REGION Network 12: Bit startu pompy w trybie awaryjnym na soft-startcie - kasowanie / Bit startu pompyw trybie awaryjnym na soft-startcie
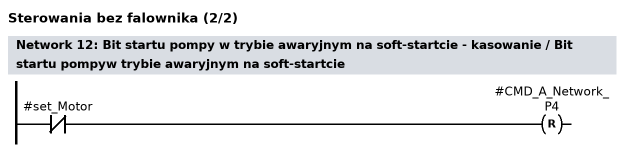
   RUNG wire#powerrail
      I_Contact( #set_Motor )
      R_Coil( #CMD_A_Network_P4 )
   END_RUNG
   // the same network as SCL:
   IF NOT #set_Motor THEN #CMD_A_Network_P4 := FALSE; END_IF;
END_REGION
END_FUNCTION_BLOCK

FUNCTION "Korekta_PV_HWrn_LWrn" : Void
TITLE = Correction
{ S7_Optimized_Access := 'TRUE' }
AUTHOR : rtecmer
VERSION : 0.1
//Funkcja wprowadza korektę ostrzerzeń wysoki i niski poziom wartości procesowej. Wartości te są następnie wykorzystane podczas sterowania pompami dodatkowymi.
   VAR_INPUT 
      PV_HWrn_correction : Real;   // Wspóczninik służący wprowadzeniu korekty ostrzeżenia przekroczenia wartości zadanej bar
      PV_LWrn_correction : Real;   // Wspóczninik służący wprowadzeniu korekty ostrzeżenia zbyt niskia wartości bar w stosunku do zadanej
   END_VAR


BEGIN
	// Funkcja pozwala na wprowadzenie korekty sygnału ostrzeżenia
	// górnrgo i dolnego wartości procesowej
	
	
	
	
	//Przetwornik błąd górny
	"dbdane"."PID_Compact_1_sPid_Cmpt.r_Pv_Hlm" := "dbtags_Sterowanie".SetupControlPompownia.r_Pv_Hlm;
	"PID_Compact_1".sPid_Cmpt.r_Pv_Hlm := "dbdane"."PID_Compact_1_sPid_Cmpt.r_Pv_Hlm";
	
	//Przetwornik błąd dolny
	"dbdane"."PID_Compact_1_sPid_Cmpt.r_Pv_Llm" := "dbtags_Sterowanie".SetupControlPompownia.r_Pv_Llm;
	"PID_Compact_1".sPid_Cmpt.r_Pv_Llm := "dbdane"."PID_Compact_1_sPid_Cmpt.r_Pv_Llm";
	
	//***Wyliczenie ostrzerzeń HWrm i LWrm ***//
	//
	"dbdane"."PID_Compact_1_sPid_Cmpt.r_Pv_HWrn" := ("db10organizacyjna".setpoint_SV_bar + #PV_HWrn_correction);
	"dbdane"."PID_Compact_1_sPid_Cmpt.r_Pv_LWrn" := ("db10organizacyjna".setpoint_SV_bar - #PV_LWrn_correction);
	
	//Ostrzegawczy wysoki
	"PID_Compact_1".sPid_Cmpt.r_Pv_HWrn := "dbdane"."PID_Compact_1_sPid_Cmpt.r_Pv_HWrn";
	"dbtags_Sterowanie".SetupControlPompownia.r_Pv_HWrn := "dbdane"."PID_Compact_1_sPid_Cmpt.r_Pv_HWrn";
	//Ostrzegawczy niski
	"PID_Compact_1".sPid_Cmpt.r_Pv_LWrn := "dbdane"."PID_Compact_1_sPid_Cmpt.r_Pv_LWrn";
	"dbtags_Sterowanie".SetupControlPompownia.r_Pv_LWrn := "dbdane"."PID_Compact_1_sPid_Cmpt.r_Pv_LWrn";
END_FUNCTION

FUNCTION "Synchroniczna_wymiana_danych_PLC1-PLC2" : Void   // FC61, LAD
TITLE = Wymiana danych
{ S7_Optimized_Access := 'TRUE' }
AUTHOR : rtecmer
VERSION : 0.1
// Funkcja grupuje bloki funkcji służąc wymianie danych HMI - PLC1, HMI-PLC2 i SCADA. Wprowadzanie wartości z poziomu HMI Zbiorniki lub HMI Pompownia czy SCADA jest nadpisywane w docelowym sterowniku. Zmian włónych parametrów układu sterowania pompownią, zbiornikami można dokonywać w dowolnego miejsca.
// stored: AutoNumber true, IsIECCheckEnabled false, SetENOAutomatically false, UDAEnableTagReadback false
   VAR_TEMP   // added for the SCL form of the ladder/FBD networks
      _w1 : Bool;
   END_VAR
BEGIN

REGION Network 2: Detekcja zmiany danych - Poziom napełnienia
   // Wymiana danych między PLC 1, PLC 2, SCADA
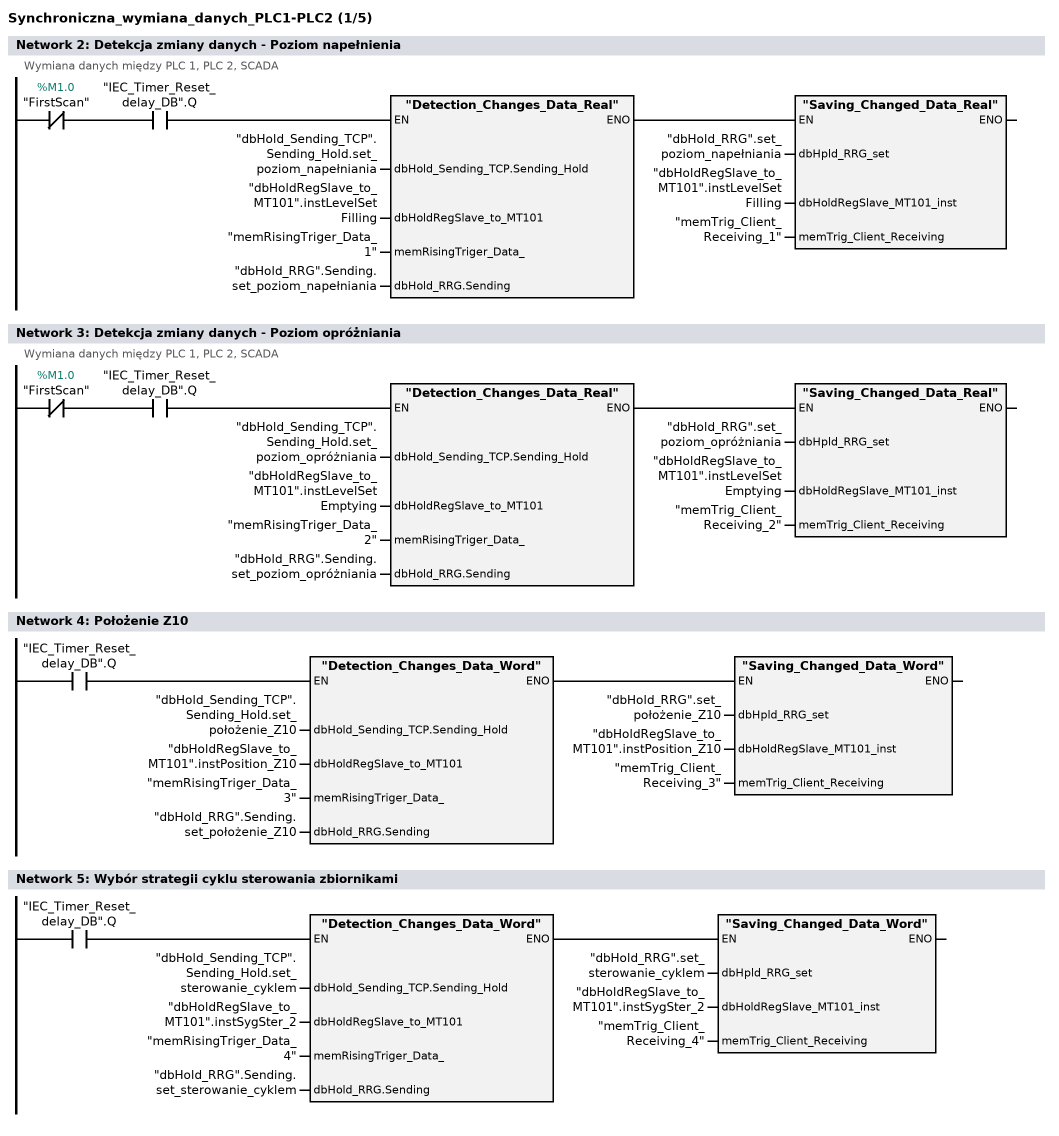
   RUNG wire#powerrail
      I_Contact( "FirstScan" )
      Contact( "IEC_Timer_Reset_delay_DB".Q )
      "Detection_Changes_Data_Real"("dbHold_Sending_TCP.Sending_Hold" := "dbHold_Sending_TCP".Sending_Hold.set_poziom_napełniania, dbHoldRegSlave_to_MT101 := "dbHoldRegSlave_to_MT101".instLevelSetFilling, memRisingTriger_Data_ := "memRisingTriger_Data_1", "dbHold_RRG.Sending" := "dbHold_RRG".Sending.set_poziom_napełniania)
      "Saving_Changed_Data_Real"(dbHpld_RRG_set := "dbHold_RRG".set_poziom_napełniania, dbHoldRegSlave_MT101_inst := "dbHoldRegSlave_to_MT101".instLevelSetFilling, memTrig_Client_Receiving := "memTrig_Client_Receiving_1")
   END_RUNG
   // the same network as SCL:
   "Detection_Changes_Data_Real"(EN := NOT "FirstScan" AND "IEC_Timer_Reset_delay_DB".Q,
                           "dbHold_Sending_TCP.Sending_Hold" := "dbHold_Sending_TCP".Sending_Hold.set_poziom_napełniania,
                           dbHoldRegSlave_to_MT101 := "dbHoldRegSlave_to_MT101".instLevelSetFilling,
                           memRisingTriger_Data_ := "memRisingTriger_Data_1",
                           "dbHold_RRG.Sending" := "dbHold_RRG".Sending.set_poziom_napełniania,
                           ENO => #_w1);
   IF #_w1 THEN
       "Saving_Changed_Data_Real"(dbHpld_RRG_set := "dbHold_RRG".set_poziom_napełniania,
                               dbHoldRegSlave_MT101_inst := "dbHoldRegSlave_to_MT101".instLevelSetFilling,
                               memTrig_Client_Receiving := "memTrig_Client_Receiving_1");
   END_IF;
END_REGION

REGION Network 3: Detekcja zmiany danych - Poziom opróżniania
   // Wymiana danych między PLC 1, PLC 2, SCADA
   RUNG wire#powerrail
      I_Contact( "FirstScan" )
      Contact( "IEC_Timer_Reset_delay_DB".Q )
      "Detection_Changes_Data_Real"("dbHold_Sending_TCP.Sending_Hold" := "dbHold_Sending_TCP".Sending_Hold.set_poziom_opróżniania, dbHoldRegSlave_to_MT101 := "dbHoldRegSlave_to_MT101".instLevelSetEmptying, memRisingTriger_Data_ := "memRisingTriger_Data_2", "dbHold_RRG.Sending" := "dbHold_RRG".Sending.set_poziom_opróżniania)
      "Saving_Changed_Data_Real"(dbHpld_RRG_set := "dbHold_RRG".set_poziom_opróżniania, dbHoldRegSlave_MT101_inst := "dbHoldRegSlave_to_MT101".instLevelSetEmptying, memTrig_Client_Receiving := "memTrig_Client_Receiving_2")
   END_RUNG
   // the same network as SCL:
   "Detection_Changes_Data_Real"(EN := NOT "FirstScan" AND "IEC_Timer_Reset_delay_DB".Q,
                           "dbHold_Sending_TCP.Sending_Hold" := "dbHold_Sending_TCP".Sending_Hold.set_poziom_opróżniania,
                           dbHoldRegSlave_to_MT101 := "dbHoldRegSlave_to_MT101".instLevelSetEmptying,
                           memRisingTriger_Data_ := "memRisingTriger_Data_2",
                           "dbHold_RRG.Sending" := "dbHold_RRG".Sending.set_poziom_opróżniania,
                           ENO => #_w1);
   IF #_w1 THEN
       "Saving_Changed_Data_Real"(dbHpld_RRG_set := "dbHold_RRG".set_poziom_opróżniania,
                               dbHoldRegSlave_MT101_inst := "dbHoldRegSlave_to_MT101".instLevelSetEmptying,
                               memTrig_Client_Receiving := "memTrig_Client_Receiving_2");
   END_IF;
END_REGION

REGION Network 4: Położenie Z10
   RUNG wire#powerrail
      Contact( "IEC_Timer_Reset_delay_DB".Q )
      "Detection_Changes_Data_Word"("dbHold_Sending_TCP.Sending_Hold" := "dbHold_Sending_TCP".Sending_Hold.set_położenie_Z10, dbHoldRegSlave_to_MT101 := "dbHoldRegSlave_to_MT101".instPosition_Z10, memRisingTriger_Data_ := "memRisingTriger_Data_3", "dbHold_RRG.Sending" := "dbHold_RRG".Sending.set_położenie_Z10)
      "Saving_Changed_Data_Word"(dbHpld_RRG_set := "dbHold_RRG".set_położenie_Z10, dbHoldRegSlave_MT101_inst := "dbHoldRegSlave_to_MT101".instPosition_Z10, memTrig_Client_Receiving := "memTrig_Client_Receiving_3")
   END_RUNG
   // the same network as SCL:
   "Detection_Changes_Data_Word"(EN := "IEC_Timer_Reset_delay_DB".Q,
                           "dbHold_Sending_TCP.Sending_Hold" := "dbHold_Sending_TCP".Sending_Hold.set_położenie_Z10,
                           dbHoldRegSlave_to_MT101 := "dbHoldRegSlave_to_MT101".instPosition_Z10,
                           memRisingTriger_Data_ := "memRisingTriger_Data_3",
                           "dbHold_RRG.Sending" := "dbHold_RRG".Sending.set_położenie_Z10,
                           ENO => #_w1);
   IF #_w1 THEN
       "Saving_Changed_Data_Word"(dbHpld_RRG_set := "dbHold_RRG".set_położenie_Z10,
                               dbHoldRegSlave_MT101_inst := "dbHoldRegSlave_to_MT101".instPosition_Z10,
                               memTrig_Client_Receiving := "memTrig_Client_Receiving_3");
   END_IF;
END_REGION

REGION Network 5: Wybór strategii cyklu sterowania zbiornikami
   RUNG wire#powerrail
      Contact( "IEC_Timer_Reset_delay_DB".Q )
      "Detection_Changes_Data_Word"("dbHold_Sending_TCP.Sending_Hold" := "dbHold_Sending_TCP".Sending_Hold.set_sterowanie_cyklem, dbHoldRegSlave_to_MT101 := "dbHoldRegSlave_to_MT101".instSygSter_2, memRisingTriger_Data_ := "memRisingTriger_Data_4", "dbHold_RRG.Sending" := "dbHold_RRG".Sending.set_sterowanie_cyklem)
      "Saving_Changed_Data_Word"(dbHpld_RRG_set := "dbHold_RRG".set_sterowanie_cyklem, dbHoldRegSlave_MT101_inst := "dbHoldRegSlave_to_MT101".instSygSter_2, memTrig_Client_Receiving := "memTrig_Client_Receiving_4")
   END_RUNG
   // the same network as SCL:
   "Detection_Changes_Data_Word"(EN := "IEC_Timer_Reset_delay_DB".Q,
                           "dbHold_Sending_TCP.Sending_Hold" := "dbHold_Sending_TCP".Sending_Hold.set_sterowanie_cyklem,
                           dbHoldRegSlave_to_MT101 := "dbHoldRegSlave_to_MT101".instSygSter_2,
                           memRisingTriger_Data_ := "memRisingTriger_Data_4",
                           "dbHold_RRG.Sending" := "dbHold_RRG".Sending.set_sterowanie_cyklem,
                           ENO => #_w1);
   IF #_w1 THEN
       "Saving_Changed_Data_Word"(dbHpld_RRG_set := "dbHold_RRG".set_sterowanie_cyklem,
                               dbHoldRegSlave_MT101_inst := "dbHoldRegSlave_to_MT101".instSygSter_2,
                               memTrig_Client_Receiving := "memTrig_Client_Receiving_4");
   END_IF;
END_REGION

REGION Network 6: Godzina napełniania start
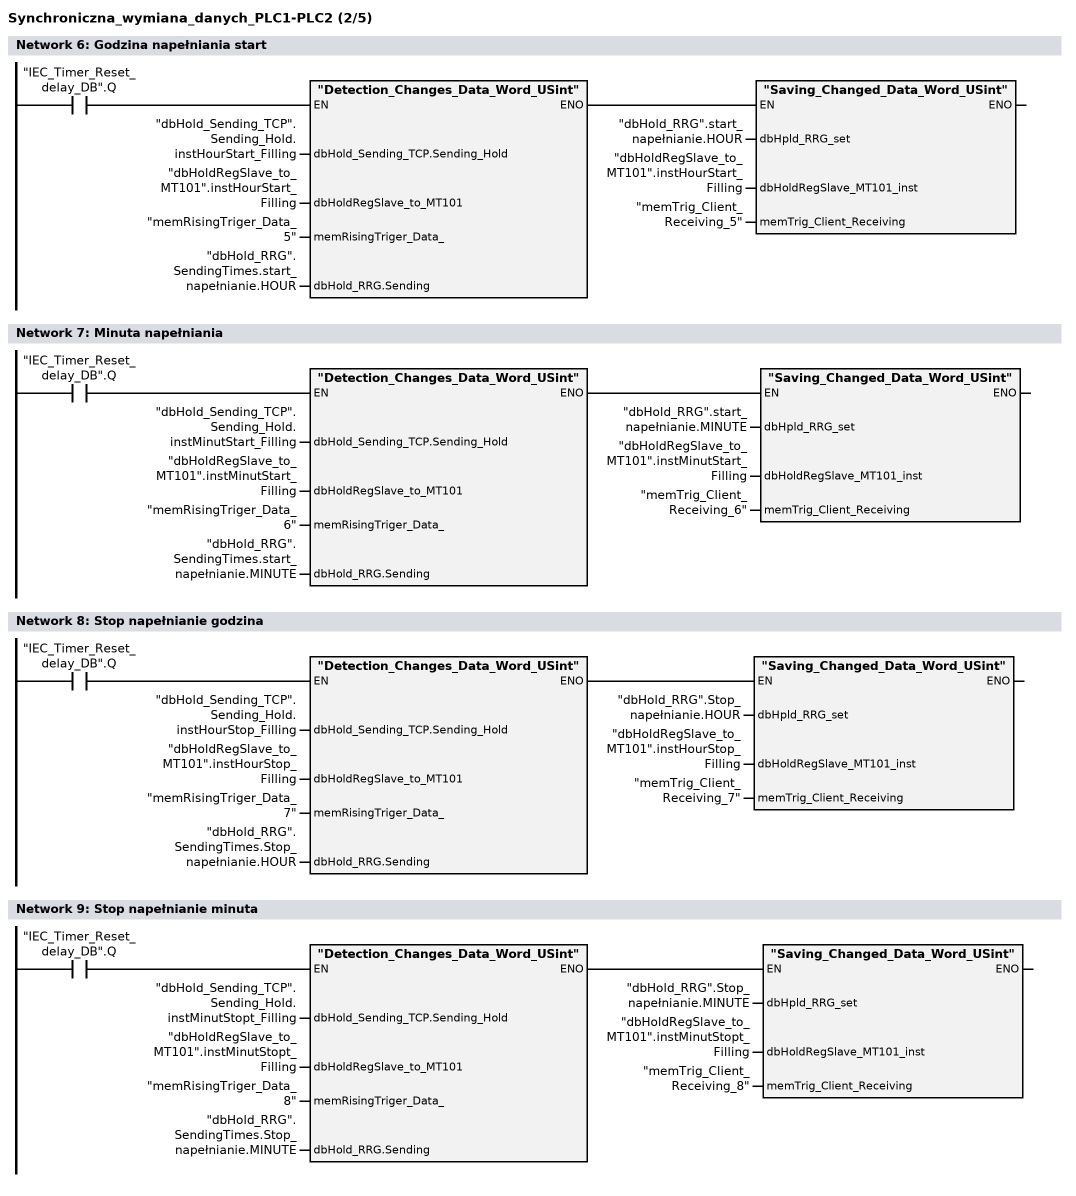
   RUNG wire#powerrail
      Contact( "IEC_Timer_Reset_delay_DB".Q )
      "Detection_Changes_Data_Word_USint"("dbHold_Sending_TCP.Sending_Hold" := "dbHold_Sending_TCP".Sending_Hold.instHourStart_Filling, dbHoldRegSlave_to_MT101 := "dbHoldRegSlave_to_MT101".instHourStart_Filling, memRisingTriger_Data_ := "memRisingTriger_Data_5", "dbHold_RRG.Sending" := "dbHold_RRG".SendingTimes.start_napełnianie.HOUR)
      "Saving_Changed_Data_Word_USint"(dbHpld_RRG_set := "dbHold_RRG".start_napełnianie.HOUR, dbHoldRegSlave_MT101_inst := "dbHoldRegSlave_to_MT101".instHourStart_Filling, memTrig_Client_Receiving := "memTrig_Client_Receiving_5")
   END_RUNG
   // the same network as SCL:
   "Detection_Changes_Data_Word_USint"(EN := "IEC_Timer_Reset_delay_DB".Q,
                           "dbHold_Sending_TCP.Sending_Hold" := "dbHold_Sending_TCP".Sending_Hold.instHourStart_Filling,
                           dbHoldRegSlave_to_MT101 := "dbHoldRegSlave_to_MT101".instHourStart_Filling,
                           memRisingTriger_Data_ := "memRisingTriger_Data_5",
                           "dbHold_RRG.Sending" := "dbHold_RRG".SendingTimes.start_napełnianie.HOUR,
                           ENO => #_w1);
   IF #_w1 THEN
       "Saving_Changed_Data_Word_USint"(dbHpld_RRG_set := "dbHold_RRG".start_napełnianie.HOUR,
                               dbHoldRegSlave_MT101_inst := "dbHoldRegSlave_to_MT101".instHourStart_Filling,
                               memTrig_Client_Receiving := "memTrig_Client_Receiving_5");
   END_IF;
END_REGION

REGION Network 7: Minuta napełniania
   RUNG wire#powerrail
      Contact( "IEC_Timer_Reset_delay_DB".Q )
      "Detection_Changes_Data_Word_USint"("dbHold_Sending_TCP.Sending_Hold" := "dbHold_Sending_TCP".Sending_Hold.instMinutStart_Filling, dbHoldRegSlave_to_MT101 := "dbHoldRegSlave_to_MT101".instMinutStart_Filling, memRisingTriger_Data_ := "memRisingTriger_Data_6", "dbHold_RRG.Sending" := "dbHold_RRG".SendingTimes.start_napełnianie.MINUTE)
      "Saving_Changed_Data_Word_USint"(dbHpld_RRG_set := "dbHold_RRG".start_napełnianie.MINUTE, dbHoldRegSlave_MT101_inst := "dbHoldRegSlave_to_MT101".instMinutStart_Filling, memTrig_Client_Receiving := "memTrig_Client_Receiving_6")
   END_RUNG
   // the same network as SCL:
   "Detection_Changes_Data_Word_USint"(EN := "IEC_Timer_Reset_delay_DB".Q,
                           "dbHold_Sending_TCP.Sending_Hold" := "dbHold_Sending_TCP".Sending_Hold.instMinutStart_Filling,
                           dbHoldRegSlave_to_MT101 := "dbHoldRegSlave_to_MT101".instMinutStart_Filling,
                           memRisingTriger_Data_ := "memRisingTriger_Data_6",
                           "dbHold_RRG.Sending" := "dbHold_RRG".SendingTimes.start_napełnianie.MINUTE,
                           ENO => #_w1);
   IF #_w1 THEN
       "Saving_Changed_Data_Word_USint"(dbHpld_RRG_set := "dbHold_RRG".start_napełnianie.MINUTE,
                               dbHoldRegSlave_MT101_inst := "dbHoldRegSlave_to_MT101".instMinutStart_Filling,
                               memTrig_Client_Receiving := "memTrig_Client_Receiving_6");
   END_IF;
END_REGION

REGION Network 8: Stop napełnianie godzina
   RUNG wire#powerrail
      Contact( "IEC_Timer_Reset_delay_DB".Q )
      "Detection_Changes_Data_Word_USint"("dbHold_Sending_TCP.Sending_Hold" := "dbHold_Sending_TCP".Sending_Hold.instHourStop_Filling, dbHoldRegSlave_to_MT101 := "dbHoldRegSlave_to_MT101".instHourStop_Filling, memRisingTriger_Data_ := "memRisingTriger_Data_7", "dbHold_RRG.Sending" := "dbHold_RRG".SendingTimes.Stop_napełnianie.HOUR)
      "Saving_Changed_Data_Word_USint"(dbHpld_RRG_set := "dbHold_RRG".Stop_napełnianie.HOUR, dbHoldRegSlave_MT101_inst := "dbHoldRegSlave_to_MT101".instHourStop_Filling, memTrig_Client_Receiving := "memTrig_Client_Receiving_7")
   END_RUNG
   // the same network as SCL:
   "Detection_Changes_Data_Word_USint"(EN := "IEC_Timer_Reset_delay_DB".Q,
                           "dbHold_Sending_TCP.Sending_Hold" := "dbHold_Sending_TCP".Sending_Hold.instHourStop_Filling,
                           dbHoldRegSlave_to_MT101 := "dbHoldRegSlave_to_MT101".instHourStop_Filling,
                           memRisingTriger_Data_ := "memRisingTriger_Data_7",
                           "dbHold_RRG.Sending" := "dbHold_RRG".SendingTimes.Stop_napełnianie.HOUR,
                           ENO => #_w1);
   IF #_w1 THEN
       "Saving_Changed_Data_Word_USint"(dbHpld_RRG_set := "dbHold_RRG".Stop_napełnianie.HOUR,
                               dbHoldRegSlave_MT101_inst := "dbHoldRegSlave_to_MT101".instHourStop_Filling,
                               memTrig_Client_Receiving := "memTrig_Client_Receiving_7");
   END_IF;
END_REGION

REGION Network 9: Stop napełnianie minuta
   RUNG wire#powerrail
      Contact( "IEC_Timer_Reset_delay_DB".Q )
      "Detection_Changes_Data_Word_USint"("dbHold_Sending_TCP.Sending_Hold" := "dbHold_Sending_TCP".Sending_Hold.instMinutStopt_Filling, dbHoldRegSlave_to_MT101 := "dbHoldRegSlave_to_MT101".instMinutStopt_Filling, memRisingTriger_Data_ := "memRisingTriger_Data_8", "dbHold_RRG.Sending" := "dbHold_RRG".SendingTimes.Stop_napełnianie.MINUTE)
      "Saving_Changed_Data_Word_USint"(dbHpld_RRG_set := "dbHold_RRG".Stop_napełnianie.MINUTE, dbHoldRegSlave_MT101_inst := "dbHoldRegSlave_to_MT101".instMinutStopt_Filling, memTrig_Client_Receiving := "memTrig_Client_Receiving_8")
   END_RUNG
   // the same network as SCL:
   "Detection_Changes_Data_Word_USint"(EN := "IEC_Timer_Reset_delay_DB".Q,
                           "dbHold_Sending_TCP.Sending_Hold" := "dbHold_Sending_TCP".Sending_Hold.instMinutStopt_Filling,
                           dbHoldRegSlave_to_MT101 := "dbHoldRegSlave_to_MT101".instMinutStopt_Filling,
                           memRisingTriger_Data_ := "memRisingTriger_Data_8",
                           "dbHold_RRG.Sending" := "dbHold_RRG".SendingTimes.Stop_napełnianie.MINUTE,
                           ENO => #_w1);
   IF #_w1 THEN
       "Saving_Changed_Data_Word_USint"(dbHpld_RRG_set := "dbHold_RRG".Stop_napełnianie.MINUTE,
                               dbHoldRegSlave_MT101_inst := "dbHoldRegSlave_to_MT101".instMinutStopt_Filling,
                               memTrig_Client_Receiving := "memTrig_Client_Receiving_8");
   END_IF;
END_REGION

REGION Network 10: Start przetłaczanie (miasto) godzina
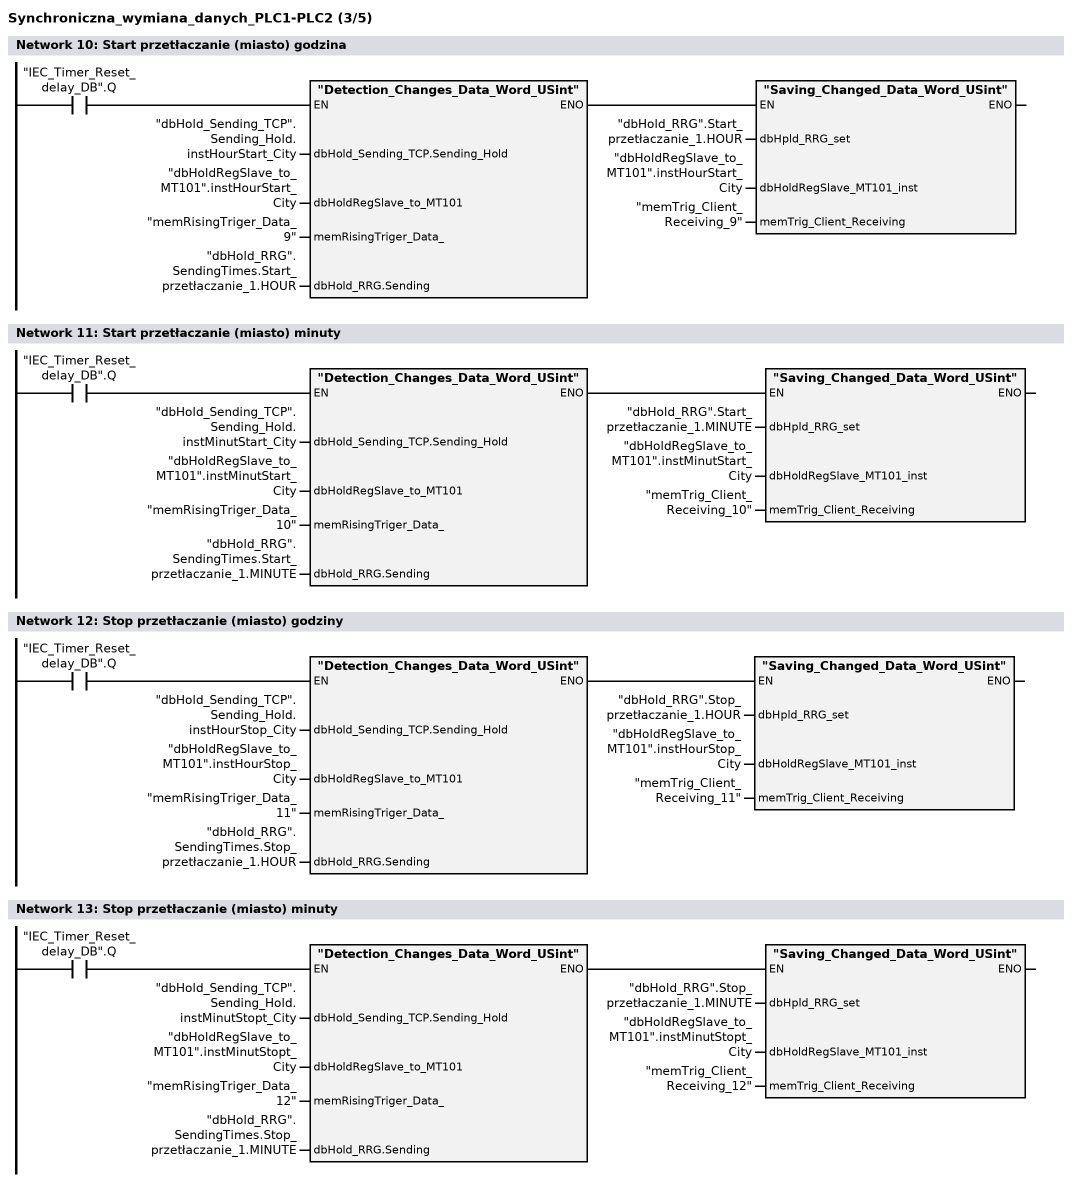
   RUNG wire#powerrail
      Contact( "IEC_Timer_Reset_delay_DB".Q )
      "Detection_Changes_Data_Word_USint"("dbHold_Sending_TCP.Sending_Hold" := "dbHold_Sending_TCP".Sending_Hold.instHourStart_City, dbHoldRegSlave_to_MT101 := "dbHoldRegSlave_to_MT101".instHourStart_City, memRisingTriger_Data_ := "memRisingTriger_Data_9", "dbHold_RRG.Sending" := "dbHold_RRG".SendingTimes.Start_przetłaczanie_1.HOUR)
      "Saving_Changed_Data_Word_USint"(dbHpld_RRG_set := "dbHold_RRG".Start_przetłaczanie_1.HOUR, dbHoldRegSlave_MT101_inst := "dbHoldRegSlave_to_MT101".instHourStart_City, memTrig_Client_Receiving := "memTrig_Client_Receiving_9")
   END_RUNG
   // the same network as SCL:
   "Detection_Changes_Data_Word_USint"(EN := "IEC_Timer_Reset_delay_DB".Q,
                           "dbHold_Sending_TCP.Sending_Hold" := "dbHold_Sending_TCP".Sending_Hold.instHourStart_City,
                           dbHoldRegSlave_to_MT101 := "dbHoldRegSlave_to_MT101".instHourStart_City,
                           memRisingTriger_Data_ := "memRisingTriger_Data_9",
                           "dbHold_RRG.Sending" := "dbHold_RRG".SendingTimes.Start_przetłaczanie_1.HOUR,
                           ENO => #_w1);
   IF #_w1 THEN
       "Saving_Changed_Data_Word_USint"(dbHpld_RRG_set := "dbHold_RRG".Start_przetłaczanie_1.HOUR,
                               dbHoldRegSlave_MT101_inst := "dbHoldRegSlave_to_MT101".instHourStart_City,
                               memTrig_Client_Receiving := "memTrig_Client_Receiving_9");
   END_IF;
END_REGION

REGION Network 11: Start przetłaczanie (miasto) minuty
   RUNG wire#powerrail
      Contact( "IEC_Timer_Reset_delay_DB".Q )
      "Detection_Changes_Data_Word_USint"("dbHold_Sending_TCP.Sending_Hold" := "dbHold_Sending_TCP".Sending_Hold.instMinutStart_City, dbHoldRegSlave_to_MT101 := "dbHoldRegSlave_to_MT101".instMinutStart_City, memRisingTriger_Data_ := "memRisingTriger_Data_10", "dbHold_RRG.Sending" := "dbHold_RRG".SendingTimes.Start_przetłaczanie_1.MINUTE)
      "Saving_Changed_Data_Word_USint"(dbHpld_RRG_set := "dbHold_RRG".Start_przetłaczanie_1.MINUTE, dbHoldRegSlave_MT101_inst := "dbHoldRegSlave_to_MT101".instMinutStart_City, memTrig_Client_Receiving := "memTrig_Client_Receiving_10")
   END_RUNG
   // the same network as SCL:
   "Detection_Changes_Data_Word_USint"(EN := "IEC_Timer_Reset_delay_DB".Q,
                           "dbHold_Sending_TCP.Sending_Hold" := "dbHold_Sending_TCP".Sending_Hold.instMinutStart_City,
                           dbHoldRegSlave_to_MT101 := "dbHoldRegSlave_to_MT101".instMinutStart_City,
                           memRisingTriger_Data_ := "memRisingTriger_Data_10",
                           "dbHold_RRG.Sending" := "dbHold_RRG".SendingTimes.Start_przetłaczanie_1.MINUTE,
                           ENO => #_w1);
   IF #_w1 THEN
       "Saving_Changed_Data_Word_USint"(dbHpld_RRG_set := "dbHold_RRG".Start_przetłaczanie_1.MINUTE,
                               dbHoldRegSlave_MT101_inst := "dbHoldRegSlave_to_MT101".instMinutStart_City,
                               memTrig_Client_Receiving := "memTrig_Client_Receiving_10");
   END_IF;
END_REGION

REGION Network 12: Stop przetłaczanie (miasto) godziny
   RUNG wire#powerrail
      Contact( "IEC_Timer_Reset_delay_DB".Q )
      "Detection_Changes_Data_Word_USint"("dbHold_Sending_TCP.Sending_Hold" := "dbHold_Sending_TCP".Sending_Hold.instHourStop_City, dbHoldRegSlave_to_MT101 := "dbHoldRegSlave_to_MT101".instHourStop_City, memRisingTriger_Data_ := "memRisingTriger_Data_11", "dbHold_RRG.Sending" := "dbHold_RRG".SendingTimes.Stop_przetłaczanie_1.HOUR)
      "Saving_Changed_Data_Word_USint"(dbHpld_RRG_set := "dbHold_RRG".Stop_przetłaczanie_1.HOUR, dbHoldRegSlave_MT101_inst := "dbHoldRegSlave_to_MT101".instHourStop_City, memTrig_Client_Receiving := "memTrig_Client_Receiving_11")
   END_RUNG
   // the same network as SCL:
   "Detection_Changes_Data_Word_USint"(EN := "IEC_Timer_Reset_delay_DB".Q,
                           "dbHold_Sending_TCP.Sending_Hold" := "dbHold_Sending_TCP".Sending_Hold.instHourStop_City,
                           dbHoldRegSlave_to_MT101 := "dbHoldRegSlave_to_MT101".instHourStop_City,
                           memRisingTriger_Data_ := "memRisingTriger_Data_11",
                           "dbHold_RRG.Sending" := "dbHold_RRG".SendingTimes.Stop_przetłaczanie_1.HOUR,
                           ENO => #_w1);
   IF #_w1 THEN
       "Saving_Changed_Data_Word_USint"(dbHpld_RRG_set := "dbHold_RRG".Stop_przetłaczanie_1.HOUR,
                               dbHoldRegSlave_MT101_inst := "dbHoldRegSlave_to_MT101".instHourStop_City,
                               memTrig_Client_Receiving := "memTrig_Client_Receiving_11");
   END_IF;
END_REGION

REGION Network 13: Stop przetłaczanie (miasto) minuty
   RUNG wire#powerrail
      Contact( "IEC_Timer_Reset_delay_DB".Q )
      "Detection_Changes_Data_Word_USint"("dbHold_Sending_TCP.Sending_Hold" := "dbHold_Sending_TCP".Sending_Hold.instMinutStopt_City, dbHoldRegSlave_to_MT101 := "dbHoldRegSlave_to_MT101".instMinutStopt_City, memRisingTriger_Data_ := "memRisingTriger_Data_12", "dbHold_RRG.Sending" := "dbHold_RRG".SendingTimes.Stop_przetłaczanie_1.MINUTE)
      "Saving_Changed_Data_Word_USint"(dbHpld_RRG_set := "dbHold_RRG".Stop_przetłaczanie_1.MINUTE, dbHoldRegSlave_MT101_inst := "dbHoldRegSlave_to_MT101".instMinutStopt_City, memTrig_Client_Receiving := "memTrig_Client_Receiving_12")
   END_RUNG
   // the same network as SCL:
   "Detection_Changes_Data_Word_USint"(EN := "IEC_Timer_Reset_delay_DB".Q,
                           "dbHold_Sending_TCP.Sending_Hold" := "dbHold_Sending_TCP".Sending_Hold.instMinutStopt_City,
                           dbHoldRegSlave_to_MT101 := "dbHoldRegSlave_to_MT101".instMinutStopt_City,
                           memRisingTriger_Data_ := "memRisingTriger_Data_12",
                           "dbHold_RRG.Sending" := "dbHold_RRG".SendingTimes.Stop_przetłaczanie_1.MINUTE,
                           ENO => #_w1);
   IF #_w1 THEN
       "Saving_Changed_Data_Word_USint"(dbHpld_RRG_set := "dbHold_RRG".Stop_przetłaczanie_1.MINUTE,
                               dbHoldRegSlave_MT101_inst := "dbHoldRegSlave_to_MT101".instMinutStopt_City,
                               memTrig_Client_Receiving := "memTrig_Client_Receiving_12");
   END_IF;
END_REGION

REGION Network 14: Start dosilanie godziny
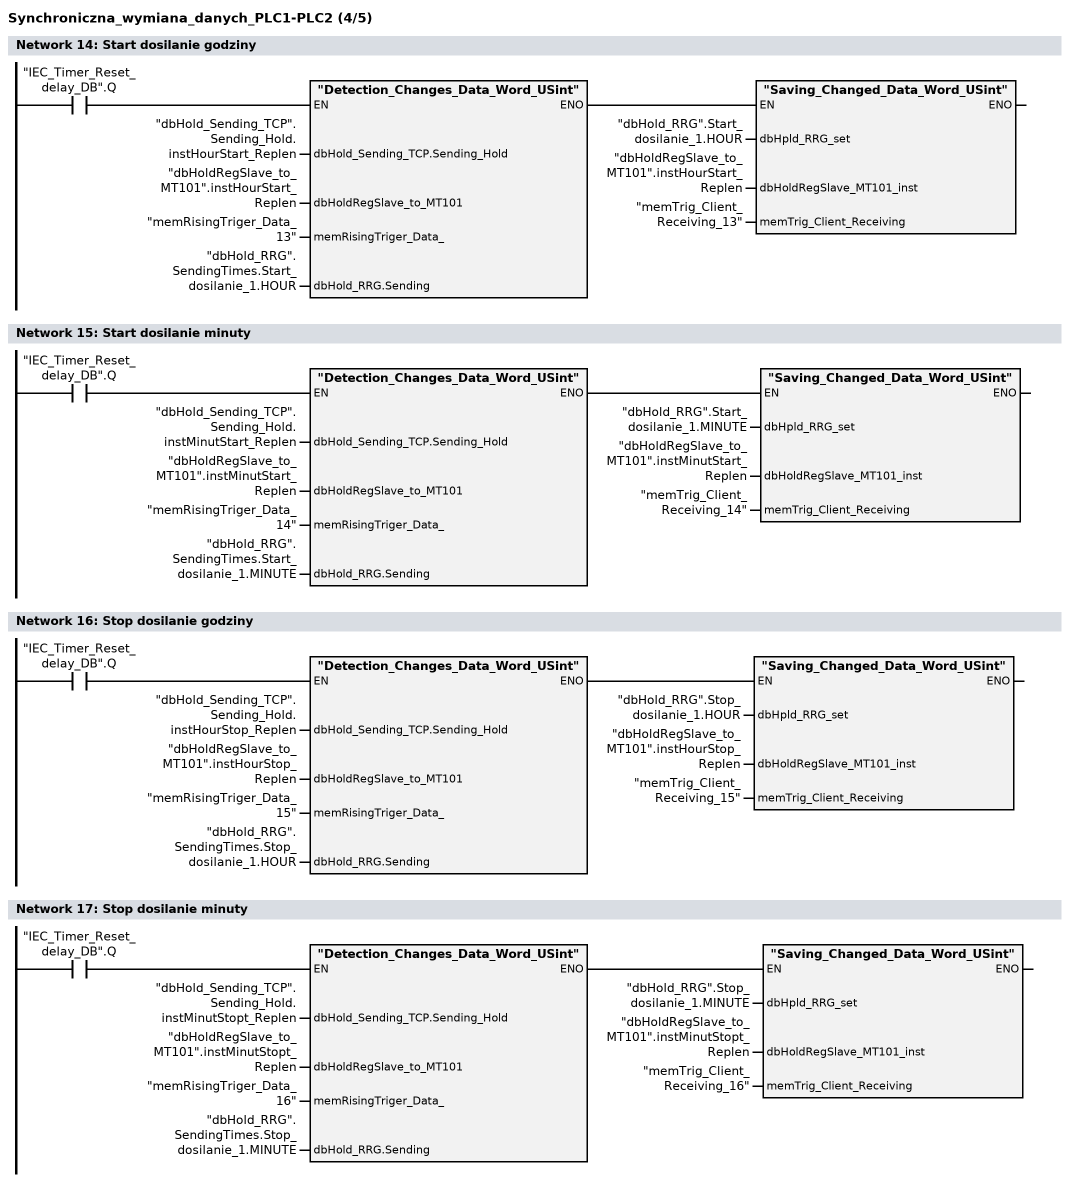
   RUNG wire#powerrail
      Contact( "IEC_Timer_Reset_delay_DB".Q )
      "Detection_Changes_Data_Word_USint"("dbHold_Sending_TCP.Sending_Hold" := "dbHold_Sending_TCP".Sending_Hold.instHourStart_Replen, dbHoldRegSlave_to_MT101 := "dbHoldRegSlave_to_MT101".instHourStart_Replen, memRisingTriger_Data_ := "memRisingTriger_Data_13", "dbHold_RRG.Sending" := "dbHold_RRG".SendingTimes.Start_dosilanie_1.HOUR)
      "Saving_Changed_Data_Word_USint"(dbHpld_RRG_set := "dbHold_RRG".Start_dosilanie_1.HOUR, dbHoldRegSlave_MT101_inst := "dbHoldRegSlave_to_MT101".instHourStart_Replen, memTrig_Client_Receiving := "memTrig_Client_Receiving_13")
   END_RUNG
   // the same network as SCL:
   "Detection_Changes_Data_Word_USint"(EN := "IEC_Timer_Reset_delay_DB".Q,
                           "dbHold_Sending_TCP.Sending_Hold" := "dbHold_Sending_TCP".Sending_Hold.instHourStart_Replen,
                           dbHoldRegSlave_to_MT101 := "dbHoldRegSlave_to_MT101".instHourStart_Replen,
                           memRisingTriger_Data_ := "memRisingTriger_Data_13",
                           "dbHold_RRG.Sending" := "dbHold_RRG".SendingTimes.Start_dosilanie_1.HOUR,
                           ENO => #_w1);
   IF #_w1 THEN
       "Saving_Changed_Data_Word_USint"(dbHpld_RRG_set := "dbHold_RRG".Start_dosilanie_1.HOUR,
                               dbHoldRegSlave_MT101_inst := "dbHoldRegSlave_to_MT101".instHourStart_Replen,
                               memTrig_Client_Receiving := "memTrig_Client_Receiving_13");
   END_IF;
END_REGION

REGION Network 15: Start dosilanie minuty
   RUNG wire#powerrail
      Contact( "IEC_Timer_Reset_delay_DB".Q )
      "Detection_Changes_Data_Word_USint"("dbHold_Sending_TCP.Sending_Hold" := "dbHold_Sending_TCP".Sending_Hold.instMinutStart_Replen, dbHoldRegSlave_to_MT101 := "dbHoldRegSlave_to_MT101".instMinutStart_Replen, memRisingTriger_Data_ := "memRisingTriger_Data_14", "dbHold_RRG.Sending" := "dbHold_RRG".SendingTimes.Start_dosilanie_1.MINUTE)
      "Saving_Changed_Data_Word_USint"(dbHpld_RRG_set := "dbHold_RRG".Start_dosilanie_1.MINUTE, dbHoldRegSlave_MT101_inst := "dbHoldRegSlave_to_MT101".instMinutStart_Replen, memTrig_Client_Receiving := "memTrig_Client_Receiving_14")
   END_RUNG
   // the same network as SCL:
   "Detection_Changes_Data_Word_USint"(EN := "IEC_Timer_Reset_delay_DB".Q,
                           "dbHold_Sending_TCP.Sending_Hold" := "dbHold_Sending_TCP".Sending_Hold.instMinutStart_Replen,
                           dbHoldRegSlave_to_MT101 := "dbHoldRegSlave_to_MT101".instMinutStart_Replen,
                           memRisingTriger_Data_ := "memRisingTriger_Data_14",
                           "dbHold_RRG.Sending" := "dbHold_RRG".SendingTimes.Start_dosilanie_1.MINUTE,
                           ENO => #_w1);
   IF #_w1 THEN
       "Saving_Changed_Data_Word_USint"(dbHpld_RRG_set := "dbHold_RRG".Start_dosilanie_1.MINUTE,
                               dbHoldRegSlave_MT101_inst := "dbHoldRegSlave_to_MT101".instMinutStart_Replen,
                               memTrig_Client_Receiving := "memTrig_Client_Receiving_14");
   END_IF;
END_REGION

REGION Network 16: Stop dosilanie godziny
   RUNG wire#powerrail
      Contact( "IEC_Timer_Reset_delay_DB".Q )
      "Detection_Changes_Data_Word_USint"("dbHold_Sending_TCP.Sending_Hold" := "dbHold_Sending_TCP".Sending_Hold.instHourStop_Replen, dbHoldRegSlave_to_MT101 := "dbHoldRegSlave_to_MT101".instHourStop_Replen, memRisingTriger_Data_ := "memRisingTriger_Data_15", "dbHold_RRG.Sending" := "dbHold_RRG".SendingTimes.Stop_dosilanie_1.HOUR)
      "Saving_Changed_Data_Word_USint"(dbHpld_RRG_set := "dbHold_RRG".Stop_dosilanie_1.HOUR, dbHoldRegSlave_MT101_inst := "dbHoldRegSlave_to_MT101".instHourStop_Replen, memTrig_Client_Receiving := "memTrig_Client_Receiving_15")
   END_RUNG
   // the same network as SCL:
   "Detection_Changes_Data_Word_USint"(EN := "IEC_Timer_Reset_delay_DB".Q,
                           "dbHold_Sending_TCP.Sending_Hold" := "dbHold_Sending_TCP".Sending_Hold.instHourStop_Replen,
                           dbHoldRegSlave_to_MT101 := "dbHoldRegSlave_to_MT101".instHourStop_Replen,
                           memRisingTriger_Data_ := "memRisingTriger_Data_15",
                           "dbHold_RRG.Sending" := "dbHold_RRG".SendingTimes.Stop_dosilanie_1.HOUR,
                           ENO => #_w1);
   IF #_w1 THEN
       "Saving_Changed_Data_Word_USint"(dbHpld_RRG_set := "dbHold_RRG".Stop_dosilanie_1.HOUR,
                               dbHoldRegSlave_MT101_inst := "dbHoldRegSlave_to_MT101".instHourStop_Replen,
                               memTrig_Client_Receiving := "memTrig_Client_Receiving_15");
   END_IF;
END_REGION

REGION Network 17: Stop dosilanie minuty
   RUNG wire#powerrail
      Contact( "IEC_Timer_Reset_delay_DB".Q )
      "Detection_Changes_Data_Word_USint"("dbHold_Sending_TCP.Sending_Hold" := "dbHold_Sending_TCP".Sending_Hold.instMinutStopt_Replen, dbHoldRegSlave_to_MT101 := "dbHoldRegSlave_to_MT101".instMinutStopt_Replen, memRisingTriger_Data_ := "memRisingTriger_Data_16", "dbHold_RRG.Sending" := "dbHold_RRG".SendingTimes.Stop_dosilanie_1.MINUTE)
      "Saving_Changed_Data_Word_USint"(dbHpld_RRG_set := "dbHold_RRG".Stop_dosilanie_1.MINUTE, dbHoldRegSlave_MT101_inst := "dbHoldRegSlave_to_MT101".instMinutStopt_Replen, memTrig_Client_Receiving := "memTrig_Client_Receiving_16")
   END_RUNG
   // the same network as SCL:
   "Detection_Changes_Data_Word_USint"(EN := "IEC_Timer_Reset_delay_DB".Q,
                           "dbHold_Sending_TCP.Sending_Hold" := "dbHold_Sending_TCP".Sending_Hold.instMinutStopt_Replen,
                           dbHoldRegSlave_to_MT101 := "dbHoldRegSlave_to_MT101".instMinutStopt_Replen,
                           memRisingTriger_Data_ := "memRisingTriger_Data_16",
                           "dbHold_RRG.Sending" := "dbHold_RRG".SendingTimes.Stop_dosilanie_1.MINUTE,
                           ENO => #_w1);
   IF #_w1 THEN
       "Saving_Changed_Data_Word_USint"(dbHpld_RRG_set := "dbHold_RRG".Stop_dosilanie_1.MINUTE,
                               dbHoldRegSlave_MT101_inst := "dbHoldRegSlave_to_MT101".instMinutStopt_Replen,
                               memTrig_Client_Receiving := "memTrig_Client_Receiving_16");
   END_IF;
END_REGION

REGION Network 19: Wybór trymu pracy M1,M2,M3,M4, Z1-Z8
   // dbHoldRegSlave_MT101 - tu wartość zadajemy 
   // dbHoldSending_TCP.Sending_Hold - z tą wzmienną porównujemy 
   // dbHold_REG.Sending - tu wysyłamy
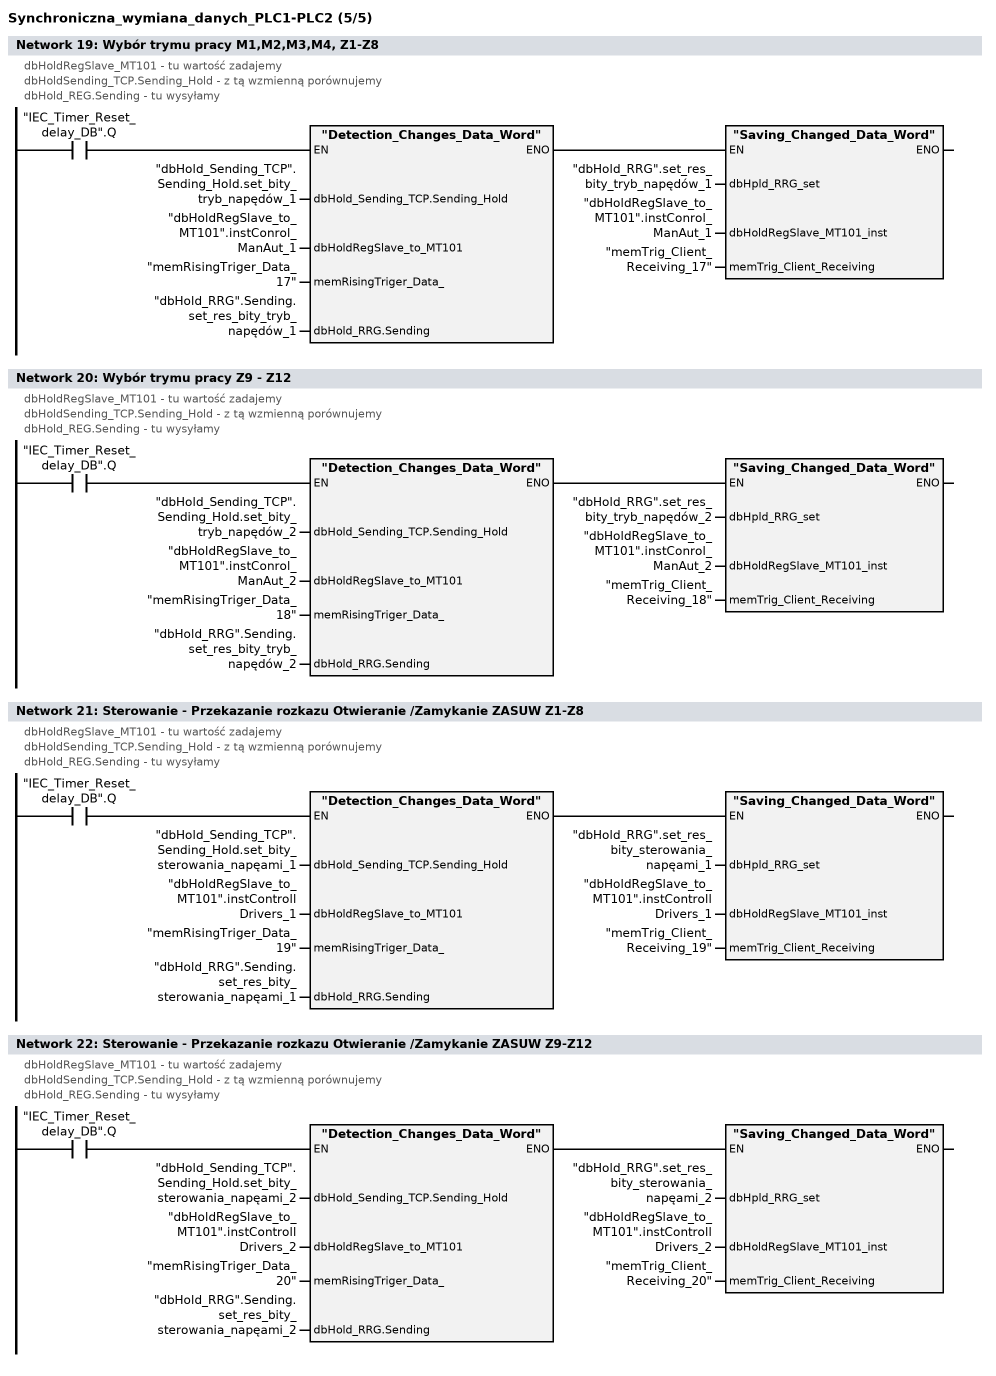
   RUNG wire#powerrail
      Contact( "IEC_Timer_Reset_delay_DB".Q )
      "Detection_Changes_Data_Word"("dbHold_Sending_TCP.Sending_Hold" := "dbHold_Sending_TCP".Sending_Hold.set_bity_tryb_napędów_1, dbHoldRegSlave_to_MT101 := "dbHoldRegSlave_to_MT101".instConrol_ManAut_1, memRisingTriger_Data_ := "memRisingTriger_Data_17", "dbHold_RRG.Sending" := "dbHold_RRG".Sending.set_res_bity_tryb_napędów_1)
      "Saving_Changed_Data_Word"(dbHpld_RRG_set := "dbHold_RRG".set_res_bity_tryb_napędów_1, dbHoldRegSlave_MT101_inst := "dbHoldRegSlave_to_MT101".instConrol_ManAut_1, memTrig_Client_Receiving := "memTrig_Client_Receiving_17")
   END_RUNG
   // the same network as SCL:
   "Detection_Changes_Data_Word"(EN := "IEC_Timer_Reset_delay_DB".Q,
                           "dbHold_Sending_TCP.Sending_Hold" := "dbHold_Sending_TCP".Sending_Hold.set_bity_tryb_napędów_1,
                           dbHoldRegSlave_to_MT101 := "dbHoldRegSlave_to_MT101".instConrol_ManAut_1,
                           memRisingTriger_Data_ := "memRisingTriger_Data_17",
                           "dbHold_RRG.Sending" := "dbHold_RRG".Sending.set_res_bity_tryb_napędów_1,
                           ENO => #_w1);
   IF #_w1 THEN
       "Saving_Changed_Data_Word"(dbHpld_RRG_set := "dbHold_RRG".set_res_bity_tryb_napędów_1,
                               dbHoldRegSlave_MT101_inst := "dbHoldRegSlave_to_MT101".instConrol_ManAut_1,
                               memTrig_Client_Receiving := "memTrig_Client_Receiving_17");
   END_IF;
END_REGION

REGION Network 20: Wybór trymu pracy Z9 - Z12
   // dbHoldRegSlave_MT101 - tu wartość zadajemy 
   // dbHoldSending_TCP.Sending_Hold - z tą wzmienną porównujemy 
   // dbHold_REG.Sending - tu wysyłamy
   RUNG wire#powerrail
      Contact( "IEC_Timer_Reset_delay_DB".Q )
      "Detection_Changes_Data_Word"("dbHold_Sending_TCP.Sending_Hold" := "dbHold_Sending_TCP".Sending_Hold.set_bity_tryb_napędów_2, dbHoldRegSlave_to_MT101 := "dbHoldRegSlave_to_MT101".instConrol_ManAut_2, memRisingTriger_Data_ := "memRisingTriger_Data_18", "dbHold_RRG.Sending" := "dbHold_RRG".Sending.set_res_bity_tryb_napędów_2)
      "Saving_Changed_Data_Word"(dbHpld_RRG_set := "dbHold_RRG".set_res_bity_tryb_napędów_2, dbHoldRegSlave_MT101_inst := "dbHoldRegSlave_to_MT101".instConrol_ManAut_2, memTrig_Client_Receiving := "memTrig_Client_Receiving_18")
   END_RUNG
   // the same network as SCL:
   "Detection_Changes_Data_Word"(EN := "IEC_Timer_Reset_delay_DB".Q,
                           "dbHold_Sending_TCP.Sending_Hold" := "dbHold_Sending_TCP".Sending_Hold.set_bity_tryb_napędów_2,
                           dbHoldRegSlave_to_MT101 := "dbHoldRegSlave_to_MT101".instConrol_ManAut_2,
                           memRisingTriger_Data_ := "memRisingTriger_Data_18",
                           "dbHold_RRG.Sending" := "dbHold_RRG".Sending.set_res_bity_tryb_napędów_2,
                           ENO => #_w1);
   IF #_w1 THEN
       "Saving_Changed_Data_Word"(dbHpld_RRG_set := "dbHold_RRG".set_res_bity_tryb_napędów_2,
                               dbHoldRegSlave_MT101_inst := "dbHoldRegSlave_to_MT101".instConrol_ManAut_2,
                               memTrig_Client_Receiving := "memTrig_Client_Receiving_18");
   END_IF;
END_REGION

REGION Network 21: Sterowanie - Przekazanie rozkazu Otwieranie /Zamykanie ZASUW Z1-Z8
   // dbHoldRegSlave_MT101 - tu wartość zadajemy 
   // dbHoldSending_TCP.Sending_Hold - z tą wzmienną porównujemy 
   // dbHold_REG.Sending - tu wysyłamy
   RUNG wire#powerrail
      Contact( "IEC_Timer_Reset_delay_DB".Q )
      "Detection_Changes_Data_Word"("dbHold_Sending_TCP.Sending_Hold" := "dbHold_Sending_TCP".Sending_Hold.set_bity_sterowania_napęami_1, dbHoldRegSlave_to_MT101 := "dbHoldRegSlave_to_MT101".instControllDrivers_1, memRisingTriger_Data_ := "memRisingTriger_Data_19", "dbHold_RRG.Sending" := "dbHold_RRG".Sending.set_res_bity_sterowania_napęami_1)
      "Saving_Changed_Data_Word"(dbHpld_RRG_set := "dbHold_RRG".set_res_bity_sterowania_napęami_1, dbHoldRegSlave_MT101_inst := "dbHoldRegSlave_to_MT101".instControllDrivers_1, memTrig_Client_Receiving := "memTrig_Client_Receiving_19")
   END_RUNG
   // the same network as SCL:
   "Detection_Changes_Data_Word"(EN := "IEC_Timer_Reset_delay_DB".Q,
                           "dbHold_Sending_TCP.Sending_Hold" := "dbHold_Sending_TCP".Sending_Hold.set_bity_sterowania_napęami_1,
                           dbHoldRegSlave_to_MT101 := "dbHoldRegSlave_to_MT101".instControllDrivers_1,
                           memRisingTriger_Data_ := "memRisingTriger_Data_19",
                           "dbHold_RRG.Sending" := "dbHold_RRG".Sending.set_res_bity_sterowania_napęami_1,
                           ENO => #_w1);
   IF #_w1 THEN
       "Saving_Changed_Data_Word"(dbHpld_RRG_set := "dbHold_RRG".set_res_bity_sterowania_napęami_1,
                               dbHoldRegSlave_MT101_inst := "dbHoldRegSlave_to_MT101".instControllDrivers_1,
                               memTrig_Client_Receiving := "memTrig_Client_Receiving_19");
   END_IF;
END_REGION

REGION Network 22: Sterowanie - Przekazanie rozkazu Otwieranie /Zamykanie ZASUW Z9-Z12
   // dbHoldRegSlave_MT101 - tu wartość zadajemy 
   // dbHoldSending_TCP.Sending_Hold - z tą wzmienną porównujemy 
   // dbHold_REG.Sending - tu wysyłamy
   RUNG wire#powerrail
      Contact( "IEC_Timer_Reset_delay_DB".Q )
      "Detection_Changes_Data_Word"("dbHold_Sending_TCP.Sending_Hold" := "dbHold_Sending_TCP".Sending_Hold.set_bity_sterowania_napęami_2, dbHoldRegSlave_to_MT101 := "dbHoldRegSlave_to_MT101".instControllDrivers_2, memRisingTriger_Data_ := "memRisingTriger_Data_20", "dbHold_RRG.Sending" := "dbHold_RRG".Sending.set_res_bity_sterowania_napęami_2)
      "Saving_Changed_Data_Word"(dbHpld_RRG_set := "dbHold_RRG".set_res_bity_sterowania_napęami_2, dbHoldRegSlave_MT101_inst := "dbHoldRegSlave_to_MT101".instControllDrivers_2, memTrig_Client_Receiving := "memTrig_Client_Receiving_20")
   END_RUNG
   // the same network as SCL:
   "Detection_Changes_Data_Word"(EN := "IEC_Timer_Reset_delay_DB".Q,
                           "dbHold_Sending_TCP.Sending_Hold" := "dbHold_Sending_TCP".Sending_Hold.set_bity_sterowania_napęami_2,
                           dbHoldRegSlave_to_MT101 := "dbHoldRegSlave_to_MT101".instControllDrivers_2,
                           memRisingTriger_Data_ := "memRisingTriger_Data_20",
                           "dbHold_RRG.Sending" := "dbHold_RRG".Sending.set_res_bity_sterowania_napęami_2,
                           ENO => #_w1);
   IF #_w1 THEN
       "Saving_Changed_Data_Word"(dbHpld_RRG_set := "dbHold_RRG".set_res_bity_sterowania_napęami_2,
                               dbHoldRegSlave_MT101_inst := "dbHoldRegSlave_to_MT101".instControllDrivers_2,
                               memTrig_Client_Receiving := "memTrig_Client_Receiving_20");
   END_IF;
END_REGION
END_FUNCTION

FUNCTION "Detection_Changes_Data_Real" : Void   // FC60, LAD
{ S7_Optimized_Access := 'TRUE' }
AUTHOR : rtecmer
VERSION : 0.1
// stored: AutoNumber true, IsIECCheckEnabled false, SetENOAutomatically false, UDAEnableTagReadback false
   VAR_IN_OUT
      "dbHold_Sending_TCP.Sending_Hold" : Real;   // Zmienna zadająca i porównywana
      dbHoldRegSlave_to_MT101 : Real;   // Zmienna w db do której porównujemy
      memRisingTriger_Data_ : Bool;   // bit pamięć zmiany
      "dbHold_RRG.Sending" : Real;   // zmienna docelowa w db do wysłania
   END_VAR
   VAR_TEMP   // added for the SCL form of the ladder/FBD networks
      _w1 : Bool;
      _w2 : Bool;
   END_VAR
BEGIN

REGION Network 1: set_poziom_napełniania
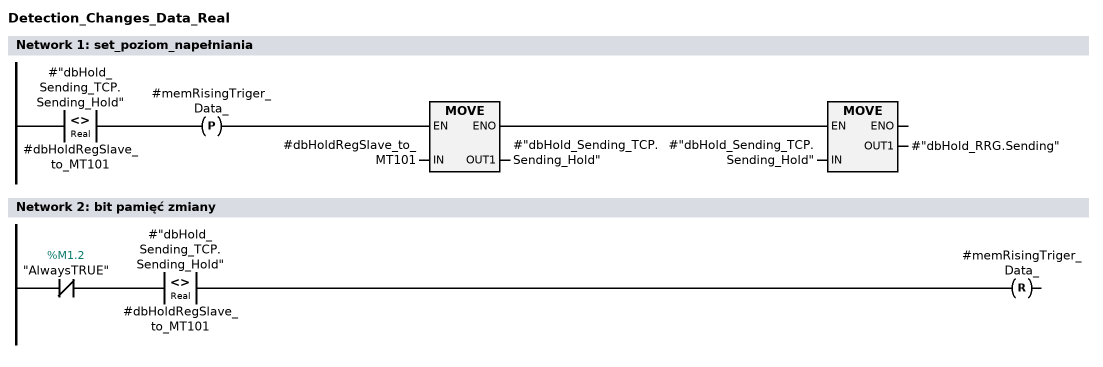
   RUNG wire#powerrail
      { S7_Templates := "SrcType := Real" } NE_Contact(in1 := #"dbHold_Sending_TCP.Sending_Hold", in2 := #dbHoldRegSlave_to_MT101)
      P_Trig( #memRisingTriger_Data_ )
      Move(in := #dbHoldRegSlave_to_MT101, out1 => #"dbHold_Sending_TCP.Sending_Hold")
      Move(in := #"dbHold_Sending_TCP.Sending_Hold", out1 => #"dbHold_RRG.Sending")
   END_RUNG
   // the same network as SCL:
   #_w1 := #"dbHold_Sending_TCP.Sending_Hold" <> #dbHoldRegSlave_to_MT101;
   #_w2 := #_w1 AND NOT #memRisingTriger_Data_;   // rising edge
   #memRisingTriger_Data_ := #_w1;
   IF #_w2 THEN
       #"dbHold_Sending_TCP.Sending_Hold" := #dbHoldRegSlave_to_MT101;
       #"dbHold_RRG.Sending" := #"dbHold_Sending_TCP.Sending_Hold";
   END_IF;
END_REGION

REGION Network 2: bit pamięć zmiany
   RUNG wire#powerrail
      I_Contact( "AlwaysTRUE" )
      { S7_Templates := "SrcType := Real" } NE_Contact(in1 := #"dbHold_Sending_TCP.Sending_Hold", in2 := #dbHoldRegSlave_to_MT101)
      R_Coil( #memRisingTriger_Data_ )
   END_RUNG
   // the same network as SCL:
   IF NOT "AlwaysTRUE" AND (#"dbHold_Sending_TCP.Sending_Hold" <> #dbHoldRegSlave_to_MT101) THEN
       #memRisingTriger_Data_ := FALSE;
   END_IF;
END_REGION
END_FUNCTION

FUNCTION "Saving_Changed_Data_Real" : Void   // FC58, LAD
{ S7_Optimized_Access := 'TRUE' }
AUTHOR : rtecmer
VERSION : 0.1
// Porównanie czy doszło do zmiany watości w db Hold_RRG <> db HoldRegSlave_toMT101
// stored: AutoNumber true, IsIECCheckEnabled false, SetENOAutomatically false, UDAEnableTagReadback false
   VAR_IN_OUT
      dbHpld_RRG_set : Real;   // Wartość zadawana porównywana
      dbHoldRegSlave_MT101_inst : Real;   // Wartość do której porównujemy
      memTrig_Client_Receiving : Bool;   // pamiec zbocza zmiany
   END_VAR
   VAR_TEMP   // added for the SCL form of the ladder/FBD networks
      _w1 : Bool;
      _w2 : Bool;
   END_VAR
BEGIN

REGION Network 1
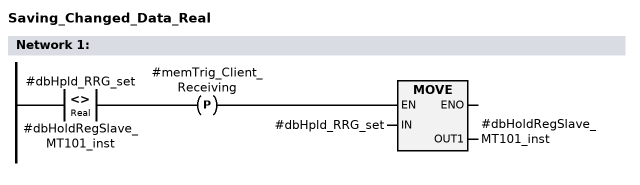
   RUNG wire#powerrail
      { S7_Templates := "SrcType := Real" } NE_Contact(in1 := #dbHpld_RRG_set, in2 := #dbHoldRegSlave_MT101_inst)
      P_Trig( #memTrig_Client_Receiving )
      Move(in := #dbHpld_RRG_set, out1 => #dbHoldRegSlave_MT101_inst)
   END_RUNG
   // the same network as SCL:
   #_w1 := #dbHpld_RRG_set <> #dbHoldRegSlave_MT101_inst;
   #_w2 := #_w1 AND NOT #memTrig_Client_Receiving;   // rising edge
   #memTrig_Client_Receiving := #_w1;
   IF #_w2 THEN #dbHoldRegSlave_MT101_inst := #dbHpld_RRG_set; END_IF;
END_REGION
END_FUNCTION

FUNCTION "Detection_Changes_Data_Word" : Void   // FC62, LAD
{ S7_Optimized_Access := 'TRUE' }
AUTHOR : rtecmer
VERSION : 0.1
// stored: AutoNumber false, IsIECCheckEnabled false, SetENOAutomatically false, UDAEnableTagReadback false
   VAR_IN_OUT
      "dbHold_Sending_TCP.Sending_Hold" : Int;   // Zmienna zadająca i porównywana
      dbHoldRegSlave_to_MT101 : Int;   // Zmienna w db do której porównujemy
      memRisingTriger_Data_ : Bool;   // bit pamięć zmiany
      "dbHold_RRG.Sending" : Int;   // zmienna docelowa w db do wysłania
   END_VAR
   VAR_TEMP   // added for the SCL form of the ladder/FBD networks
      _w1 : Bool;
      _w2 : Bool;
   END_VAR
BEGIN

REGION Network 1: set_poziom_napełniania
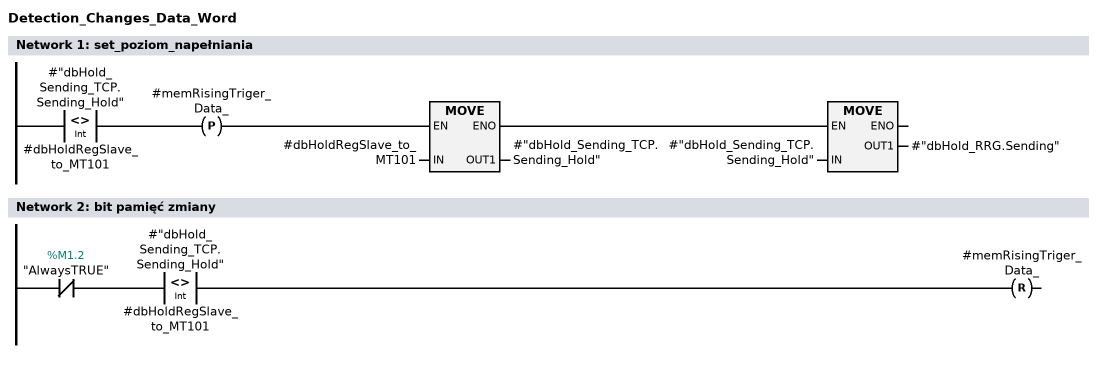
   RUNG wire#powerrail
      { S7_Templates := "SrcType := Int" } NE_Contact(in1 := #"dbHold_Sending_TCP.Sending_Hold", in2 := #dbHoldRegSlave_to_MT101)
      P_Trig( #memRisingTriger_Data_ )
      Move(in := #dbHoldRegSlave_to_MT101, out1 => #"dbHold_Sending_TCP.Sending_Hold")
      Move(in := #"dbHold_Sending_TCP.Sending_Hold", out1 => #"dbHold_RRG.Sending")
   END_RUNG
   // the same network as SCL:
   #_w1 := #"dbHold_Sending_TCP.Sending_Hold" <> #dbHoldRegSlave_to_MT101;
   #_w2 := #_w1 AND NOT #memRisingTriger_Data_;   // rising edge
   #memRisingTriger_Data_ := #_w1;
   IF #_w2 THEN
       #"dbHold_Sending_TCP.Sending_Hold" := #dbHoldRegSlave_to_MT101;
       #"dbHold_RRG.Sending" := #"dbHold_Sending_TCP.Sending_Hold";
   END_IF;
END_REGION

REGION Network 2: bit pamięć zmiany
   RUNG wire#powerrail
      I_Contact( "AlwaysTRUE" )
      { S7_Templates := "SrcType := Int" } NE_Contact(in1 := #"dbHold_Sending_TCP.Sending_Hold", in2 := #dbHoldRegSlave_to_MT101)
      R_Coil( #memRisingTriger_Data_ )
   END_RUNG
   // the same network as SCL:
   IF NOT "AlwaysTRUE" AND (#"dbHold_Sending_TCP.Sending_Hold" <> #dbHoldRegSlave_to_MT101) THEN
       #memRisingTriger_Data_ := FALSE;
   END_IF;
END_REGION
END_FUNCTION

FUNCTION "Saving_Changed_Data_Word" : Void   // FC59, LAD
{ S7_Optimized_Access := 'TRUE' }
AUTHOR : rtecmer
VERSION : 0.1
// Porównanie czy doszło do zmiany watości w db Hold_RRG <> db HoldRegSlave_toMT101
// stored: AutoNumber false, IsIECCheckEnabled false, SetENOAutomatically false, UDAEnableTagReadback false
   VAR_IN_OUT
      dbHpld_RRG_set : Int;   // Wartość zadawana porównywana
      dbHoldRegSlave_MT101_inst : Int;   // Wartość do której porównujemy
      memTrig_Client_Receiving : Bool;   // pamiec zbocza zmiany
   END_VAR
   VAR_TEMP   // added for the SCL form of the ladder/FBD networks
      _w1 : Bool;
      _w2 : Bool;
   END_VAR
BEGIN

REGION Network 1
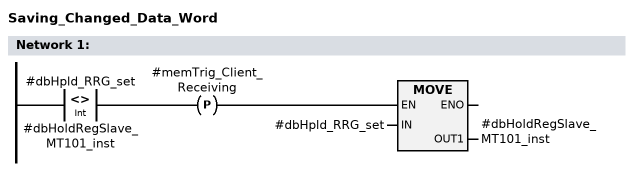
   RUNG wire#powerrail
      { S7_Templates := "SrcType := Int" } NE_Contact(in1 := #dbHpld_RRG_set, in2 := #dbHoldRegSlave_MT101_inst)
      P_Trig( #memTrig_Client_Receiving )
      Move(in := #dbHpld_RRG_set, out1 => #dbHoldRegSlave_MT101_inst)
   END_RUNG
   // the same network as SCL:
   #_w1 := #dbHpld_RRG_set <> #dbHoldRegSlave_MT101_inst;
   #_w2 := #_w1 AND NOT #memTrig_Client_Receiving;   // rising edge
   #memTrig_Client_Receiving := #_w1;
   IF #_w2 THEN #dbHoldRegSlave_MT101_inst := #dbHpld_RRG_set; END_IF;
END_REGION
END_FUNCTION

FUNCTION "Detection_Changes_Data_Word_USint" : Void   // FC64, LAD
{ S7_Optimized_Access := 'TRUE' }
AUTHOR : rtecmer
VERSION : 0.1
// stored: AutoNumber false, IsIECCheckEnabled false, SetENOAutomatically false, UDAEnableTagReadback false
   VAR_IN_OUT
      "dbHold_Sending_TCP.Sending_Hold" : Int;   // Zmienna zadająca i porównywana
      dbHoldRegSlave_to_MT101 : Int;   // Zmienna w db do której porównujemy
      memRisingTriger_Data_ : Bool;   // bit pamięć zmiany
      "dbHold_RRG.Sending" : USInt;   // zmienna docelowa w db do wysłania
   END_VAR
   VAR_TEMP   // added for the SCL form of the ladder/FBD networks
      _w1 : Bool;
      _w2 : Bool;
   END_VAR
BEGIN

REGION Network 1: set_poziom_napełniania
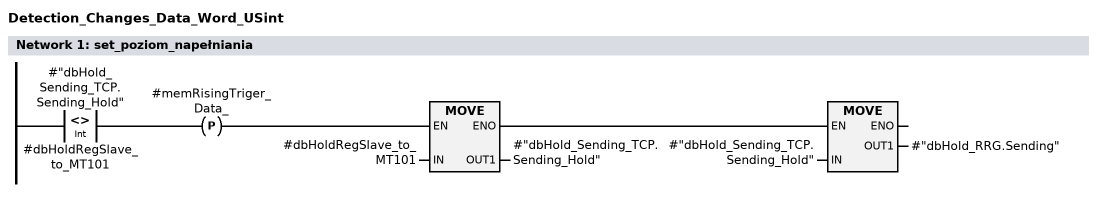
   RUNG wire#powerrail
      { S7_Templates := "SrcType := Int" } NE_Contact(in1 := #"dbHold_Sending_TCP.Sending_Hold", in2 := #dbHoldRegSlave_to_MT101)
      P_Trig( #memRisingTriger_Data_ )
      Move(in := #dbHoldRegSlave_to_MT101, out1 => #"dbHold_Sending_TCP.Sending_Hold")
      Move(in := #"dbHold_Sending_TCP.Sending_Hold", out1 => #"dbHold_RRG.Sending")
   END_RUNG
   // the same network as SCL:
   #_w1 := #"dbHold_Sending_TCP.Sending_Hold" <> #dbHoldRegSlave_to_MT101;
   #_w2 := #_w1 AND NOT #memRisingTriger_Data_;   // rising edge
   #memRisingTriger_Data_ := #_w1;
   IF #_w2 THEN
       #"dbHold_Sending_TCP.Sending_Hold" := #dbHoldRegSlave_to_MT101;
       #"dbHold_RRG.Sending" := #"dbHold_Sending_TCP.Sending_Hold";
   END_IF;
END_REGION
END_FUNCTION

FUNCTION "Saving_Changed_Data_Word_USint" : Void   // FC65, LAD
{ S7_Optimized_Access := 'TRUE' }
AUTHOR : rtecmer
VERSION : 0.1
// Porównanie czy doszło do zmiany watości w db Hold_RRG <> db HoldRegSlave_toMT101
// stored: AutoNumber false, IsIECCheckEnabled false, SetENOAutomatically false, UDAEnableTagReadback false
   VAR_IN_OUT
      dbHpld_RRG_set : USInt;   // Wartość zadawana porównywana
      dbHoldRegSlave_MT101_inst : Int;   // Wartość do której porównujemy
      memTrig_Client_Receiving : Bool;   // pamiec zbocza zmiany
   END_VAR
   VAR_TEMP   // added for the SCL form of the ladder/FBD networks
      _w1 : Bool;
      _w2 : Bool;
   END_VAR
BEGIN

REGION Network 1
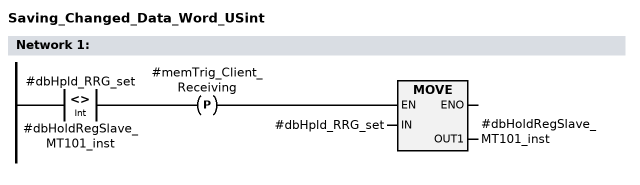
   RUNG wire#powerrail
      { S7_Templates := "SrcType := Int" } NE_Contact(in1 := #dbHpld_RRG_set, in2 := #dbHoldRegSlave_MT101_inst)
      P_Trig( #memTrig_Client_Receiving )
      Move(in := #dbHpld_RRG_set, out1 => #dbHoldRegSlave_MT101_inst)
   END_RUNG
   // the same network as SCL:
   #_w1 := #dbHpld_RRG_set <> #dbHoldRegSlave_MT101_inst;
   #_w2 := #_w1 AND NOT #memTrig_Client_Receiving;   // rising edge
   #memTrig_Client_Receiving := #_w1;
   IF #_w2 THEN #dbHoldRegSlave_MT101_inst := #dbHpld_RRG_set; END_IF;
END_REGION
END_FUNCTION

FUNCTION "Sterownik_P1P2P3P4" : Void   // FC3, LAD
{ S7_Optimized_Access := 'TRUE' }
AUTHOR : RTecmer
VERSION : 0.1
// Sterowaniepompownią
// Funkcja zarządza sygnałem załączającym styczniki (sieć), (Falownik) danego napędu
// Sterowanie kompresorami
// Algorytm przewiduje sterowanie nadrzędne w trybie automatycznym przez sterownik master "OMROM". Sterowanie w trybie Manual z systemu SCADA odbywa się przez sterownik SLAVE "S7-1200" . Sterownik S7-100 reguluje sygnałem zadawania Hz w oparciu o regulator PID. Sygnał ten podawany jest na wejście analogowe sterownika Master. Praca sterownika S7-1200 Slave ogranicza się do generowania sygnału Hz, wystawianiu sygnału Automat, sygnału Dodatkowy kompresor 1, sygnału Dodatkowy kompresor 2. Komunikacji z systemem SCADA.
// stored: AutoNumber true, IsIECCheckEnabled false, SetENOAutomatically false, UDAEnableTagReadback false
BEGIN

REGION Network 1: Drive P1 / P1 Driver
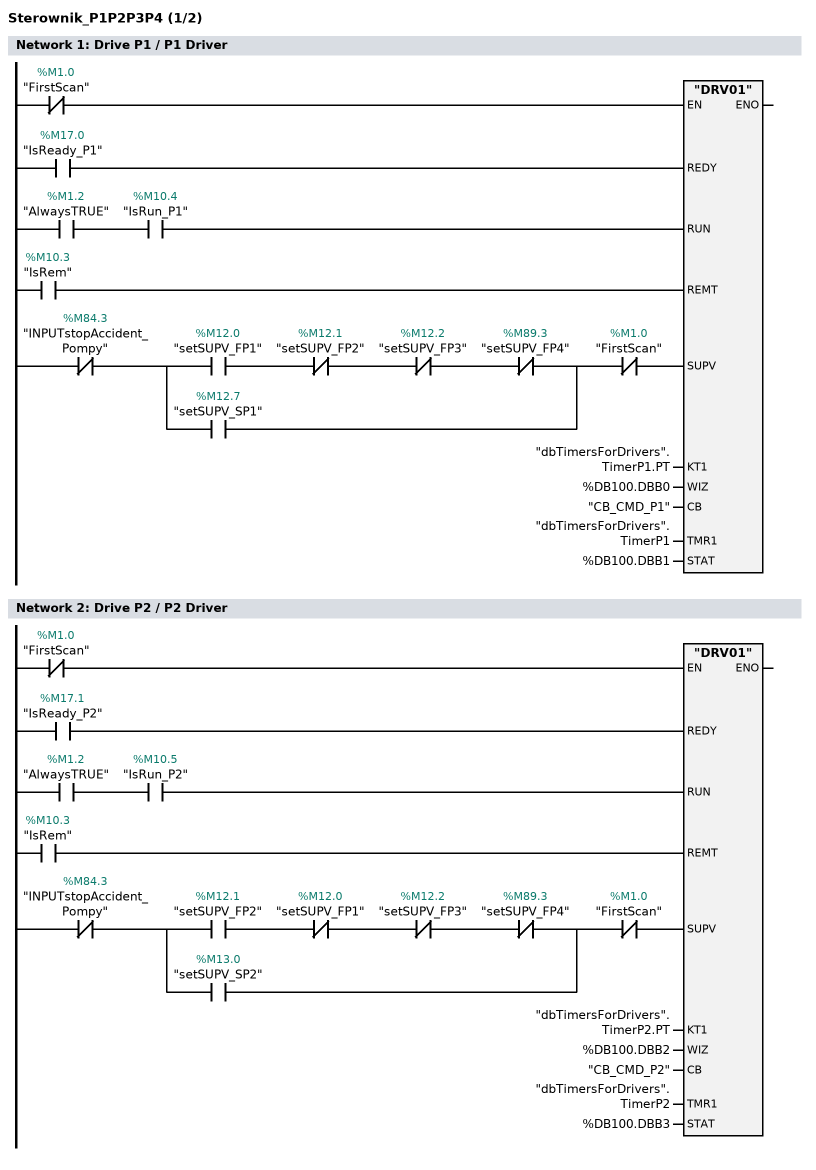
   RUNG wire#powerrail
      I_Contact( "FirstScan" )
      "DRV01"(REDY := wire#w1, RUN := wire#w2, REMT := wire#w3, SUPV := wire#w6, KT1 := "dbTimersForDrivers".TimerP1.PT, WIZ := %DB100.DBB0, CB := "CB_CMD_P1", TMR1 := "dbTimersForDrivers".TimerP1, STAT := %DB100.DBB1)
   END_RUNG
   RUNG wire#powerrail
      Contact( "IsReady_P1" )
   END_RUNG wire#w1
   RUNG wire#powerrail
      Contact( "AlwaysTRUE" )
      Contact( "IsRun_P1" )
   END_RUNG wire#w2
   RUNG wire#powerrail
      Contact( "IsRem" )
   END_RUNG wire#w3
   RUNG wire#powerrail
      I_Contact( "INPUTstopAccident_Pompy" )
      wire#w4
      Contact( "setSUPV_FP1" )
      I_Contact( "setSUPV_FP2" )
      I_Contact( "setSUPV_FP3" )
      I_Contact( "setSUPV_FP4" )
      wire#w5
      I_Contact( "FirstScan" )
   END_RUNG wire#w6
   RUNG wire#w4
      Contact( "setSUPV_SP1" )
   END_RUNG wire#w5
   // the same network as SCL:
   IF NOT "FirstScan" THEN
       "DRV01"(REDY := "IsReady_P1",
               RUN := "AlwaysTRUE" AND "IsRun_P1",
               REMT := "IsRem",
               SUPV := NOT "INPUTstopAccident_Pompy" AND (("setSUPV_FP1" AND NOT "setSUPV_FP2" AND NOT "setSUPV_FP3" AND NOT "setSUPV_FP4") OR "setSUPV_SP1") AND NOT "FirstScan",
               KT1 := "dbTimersForDrivers".TimerP1.PT,
               WIZ := %DB100.DBB0,
               CB := "CB_CMD_P1",
               TMR1 := "dbTimersForDrivers".TimerP1,
               STAT := %DB100.DBB1);
   END_IF;
END_REGION

REGION Network 2: Drive P2 / P2 Driver
   RUNG wire#powerrail
      I_Contact( "FirstScan" )
      "DRV01"(REDY := wire#w1, RUN := wire#w2, REMT := wire#w3, SUPV := wire#w6, KT1 := "dbTimersForDrivers".TimerP2.PT, WIZ := %DB100.DBB2, CB := "CB_CMD_P2", TMR1 := "dbTimersForDrivers".TimerP2, STAT := %DB100.DBB3)
   END_RUNG
   RUNG wire#powerrail
      Contact( "IsReady_P2" )
   END_RUNG wire#w1
   RUNG wire#powerrail
      Contact( "AlwaysTRUE" )
      Contact( "IsRun_P2" )
   END_RUNG wire#w2
   RUNG wire#powerrail
      Contact( "IsRem" )
   END_RUNG wire#w3
   RUNG wire#powerrail
      I_Contact( "INPUTstopAccident_Pompy" )
      wire#w4
      Contact( "setSUPV_FP2" )
      I_Contact( "setSUPV_FP1" )
      I_Contact( "setSUPV_FP3" )
      I_Contact( "setSUPV_FP4" )
      wire#w5
      I_Contact( "FirstScan" )
   END_RUNG wire#w6
   RUNG wire#w4
      Contact( "setSUPV_SP2" )
   END_RUNG wire#w5
   // the same network as SCL:
   IF NOT "FirstScan" THEN
       "DRV01"(REDY := "IsReady_P2",
               RUN := "AlwaysTRUE" AND "IsRun_P2",
               REMT := "IsRem",
               SUPV := NOT "INPUTstopAccident_Pompy" AND (("setSUPV_FP2" AND NOT "setSUPV_FP1" AND NOT "setSUPV_FP3" AND NOT "setSUPV_FP4") OR "setSUPV_SP2") AND NOT "FirstScan",
               KT1 := "dbTimersForDrivers".TimerP2.PT,
               WIZ := %DB100.DBB2,
               CB := "CB_CMD_P2",
               TMR1 := "dbTimersForDrivers".TimerP2,
               STAT := %DB100.DBB3);
   END_IF;
END_REGION

REGION Network 3: Drive P3 / P3 Driver
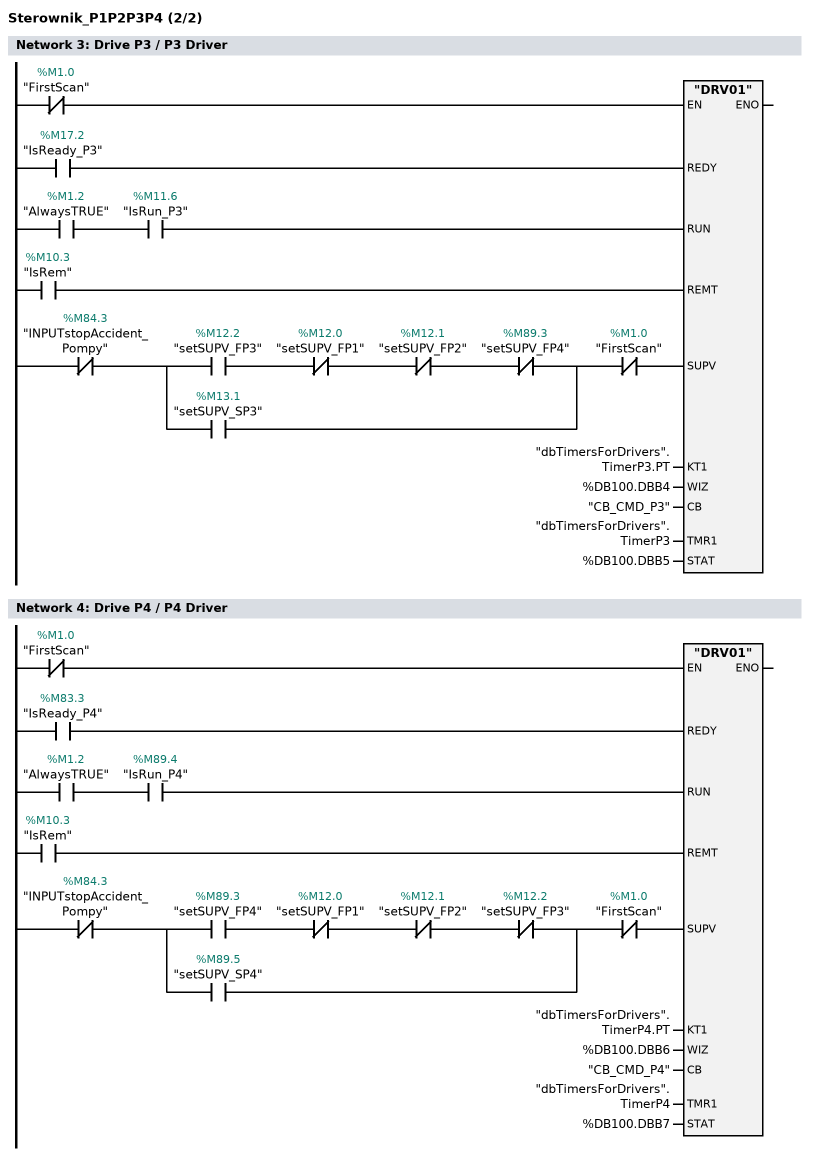
   RUNG wire#powerrail
      I_Contact( "FirstScan" )
      "DRV01"(REDY := wire#w1, RUN := wire#w2, REMT := wire#w3, SUPV := wire#w6, KT1 := "dbTimersForDrivers".TimerP3.PT, WIZ := %DB100.DBB4, CB := "CB_CMD_P3", TMR1 := "dbTimersForDrivers".TimerP3, STAT := %DB100.DBB5)
   END_RUNG
   RUNG wire#powerrail
      Contact( "IsReady_P3" )
   END_RUNG wire#w1
   RUNG wire#powerrail
      Contact( "AlwaysTRUE" )
      Contact( "IsRun_P3" )
   END_RUNG wire#w2
   RUNG wire#powerrail
      Contact( "IsRem" )
   END_RUNG wire#w3
   RUNG wire#powerrail
      I_Contact( "INPUTstopAccident_Pompy" )
      wire#w4
      Contact( "setSUPV_FP3" )
      I_Contact( "setSUPV_FP1" )
      I_Contact( "setSUPV_FP2" )
      I_Contact( "setSUPV_FP4" )
      wire#w5
      I_Contact( "FirstScan" )
   END_RUNG wire#w6
   RUNG wire#w4
      Contact( "setSUPV_SP3" )
   END_RUNG wire#w5
   // the same network as SCL:
   IF NOT "FirstScan" THEN
       "DRV01"(REDY := "IsReady_P3",
               RUN := "AlwaysTRUE" AND "IsRun_P3",
               REMT := "IsRem",
               SUPV := NOT "INPUTstopAccident_Pompy" AND (("setSUPV_FP3" AND NOT "setSUPV_FP1" AND NOT "setSUPV_FP2" AND NOT "setSUPV_FP4") OR "setSUPV_SP3") AND NOT "FirstScan",
               KT1 := "dbTimersForDrivers".TimerP3.PT,
               WIZ := %DB100.DBB4,
               CB := "CB_CMD_P3",
               TMR1 := "dbTimersForDrivers".TimerP3,
               STAT := %DB100.DBB5);
   END_IF;
END_REGION

REGION Network 4: Drive P4 / P4 Driver
   RUNG wire#powerrail
      I_Contact( "FirstScan" )
      "DRV01"(REDY := wire#w1, RUN := wire#w2, REMT := wire#w3, SUPV := wire#w6, KT1 := "dbTimersForDrivers".TimerP4.PT, WIZ := %DB100.DBB6, CB := "CB_CMD_P4", TMR1 := "dbTimersForDrivers".TimerP4, STAT := %DB100.DBB7)
   END_RUNG
   RUNG wire#powerrail
      Contact( "IsReady_P4" )
   END_RUNG wire#w1
   RUNG wire#powerrail
      Contact( "AlwaysTRUE" )
      Contact( "IsRun_P4" )
   END_RUNG wire#w2
   RUNG wire#powerrail
      Contact( "IsRem" )
   END_RUNG wire#w3
   RUNG wire#powerrail
      I_Contact( "INPUTstopAccident_Pompy" )
      wire#w4
      Contact( "setSUPV_FP4" )
      I_Contact( "setSUPV_FP1" )
      I_Contact( "setSUPV_FP2" )
      I_Contact( "setSUPV_FP3" )
      wire#w5
      I_Contact( "FirstScan" )
   END_RUNG wire#w6
   RUNG wire#w4
      Contact( "setSUPV_SP4" )
   END_RUNG wire#w5
   // the same network as SCL:
   IF NOT "FirstScan" THEN
       "DRV01"(REDY := "IsReady_P4",
               RUN := "AlwaysTRUE" AND "IsRun_P4",
               REMT := "IsRem",
               SUPV := NOT "INPUTstopAccident_Pompy" AND (("setSUPV_FP4" AND NOT "setSUPV_FP1" AND NOT "setSUPV_FP2" AND NOT "setSUPV_FP3") OR "setSUPV_SP4") AND NOT "FirstScan",
               KT1 := "dbTimersForDrivers".TimerP4.PT,
               WIZ := %DB100.DBB6,
               CB := "CB_CMD_P4",
               TMR1 := "dbTimersForDrivers".TimerP4,
               STAT := %DB100.DBB7);
   END_IF;
END_REGION
END_FUNCTION

FUNCTION "DRV01" : Void   // FC1, LAD
TITLE = Funkcja sterowania stycznikiem silnika
{ S7_Optimized_Access := 'FALSE' }
VERSION : 0.1
// Funkcja standardowa sluzy do zalaczania silnika.
// Posiada trzy tryby pracy:
//      - localny (zalaczanie  elektrycznie bez PLC)
//      - zdalny  (zalaczanie przez PLC)
//          - reczny (zalaczanie przez dyspozytora z SCADA)
//          - automatyczny (zalaczanie wynikle z algotytmu sterowania)
// Zrodlo danych dla funkcji stanowia:
//      - sygnaly I/O PLC
//          - =REDY -gotowosc napedu
//          - =REMT -sterowanie napedu 1-zdalnie 0-local
//          - =RUN  -naped wlaczony
//          - =CB   -zalaczenie stycznika
//       - =STAT bajt statusu napedu 
//               jego kopia w DB =WIZ stanowi interface PLC/MMI
//          - bit 0 Alarm              (sygnal do MMI)
//          - bit 1  
//          - bit 2 kopia sygnalu REMT (sygnal do SCADA)
//          - bit 3 kopia sygnalu RUN  (sygnal do SCADA)
//          - bit 4 wylaczenie reczne  (sygnal z SCADA) 
//          - bit 5 wlaczenie reczne   (sygnal z SCADA)
//          - bit 6 alarm reset        (sygnal z SCADA)
//          - bit 7 1=auto, 0=man      (sygnal z SCADA)
//        - =SUPV - sygnal zalacznia w trybie automatycznym
//        - sygnaly czasowe
//          - =TMR1 -kontrola czasu zalaczenia stycznika
//          - =KT1  -wartosc czasu timera 1
//          - flagi
// stored: AutoNumber false, IsIECCheckEnabled false, SetENOAutomatically false, UDAEnableTagReadback false
   VAR_INPUT
      REDY : Bool;   // Sygnał gotowości
      RUN : Bool;   // Sygnał pracy
      REMT : Bool;   // Sterowanie napędu zdalne-1 lokalne -0
      SUPV : Bool;   // Sygnalizacja załączenia w trybie automatycznym
      KT1 : Time;   // wartosc czasu timera 1
   END_VAR
   VAR_IN_OUT
      WIZ : Byte;   // Wektor stanu ze SCADA
      CB : Bool;   // Przekaźnik urządzenia
      TMR1 : TON_TIME;   // Kontrola czasu załączenia stycznika
      STAT : Byte;   // Wektor stanu urządzenia
   END_VAR
   // Ret_Val : Napęd jednokierunkowy - pompy
BEGIN

REGION Network 1: Network 1: mapowanie wektora statusu napędu i stanu wektora z SCADA
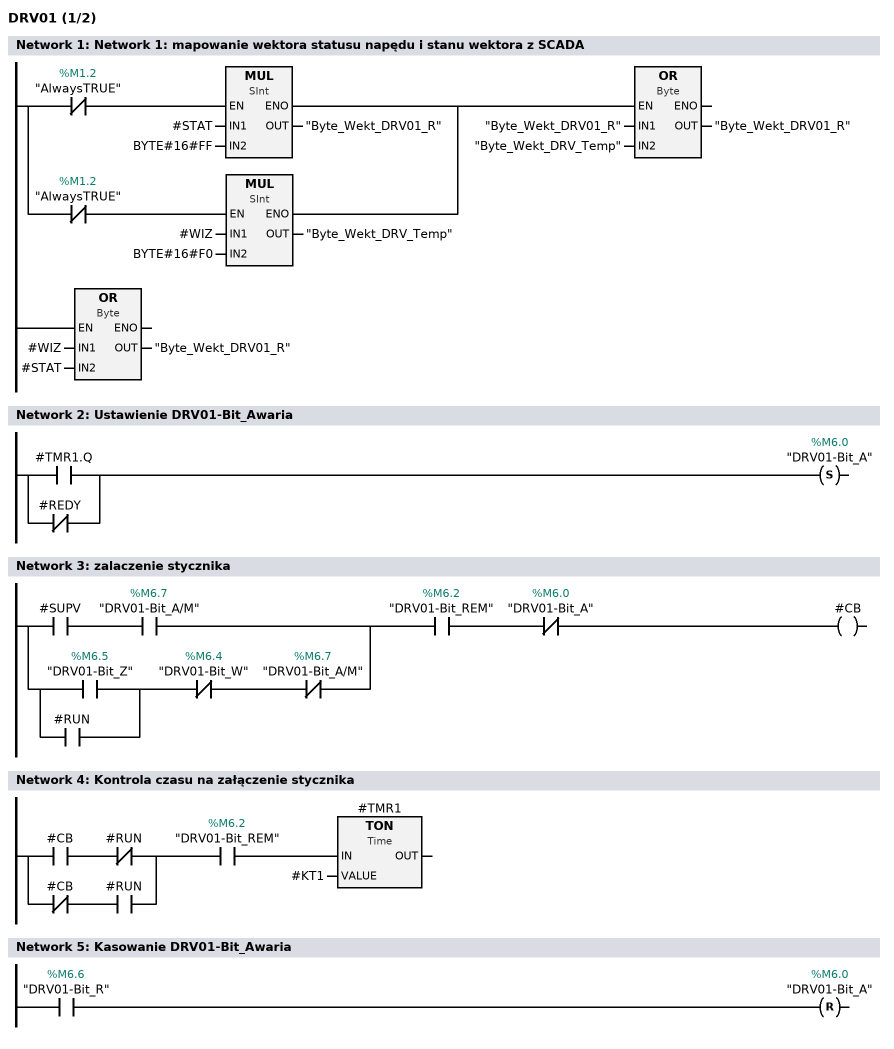
   // ENO of a box is taken as its EN; it also drops when the box reports an error
   IF NOT "AlwaysTRUE" THEN
       "Byte_Wekt_DRV01_R" := #STAT * BYTE#16#FF;
       "Byte_Wekt_DRV_Temp" := #WIZ * BYTE#16#F0;
   END_IF;
   IF NOT "AlwaysTRUE" OR NOT "AlwaysTRUE" THEN
       "Byte_Wekt_DRV01_R" := "Byte_Wekt_DRV01_R" OR "Byte_Wekt_DRV_Temp";
   END_IF;
   "Byte_Wekt_DRV01_R" := #WIZ OR #STAT;
END_REGION

REGION Network 2: Ustawienie DRV01-Bit_Awaria
   RUNG wire#powerrail
      Contact( #TMR1.Q )
      wire#w1
      S_Coil( "DRV01-Bit_A" )
   END_RUNG
   RUNG wire#powerrail
      I_Contact( #REDY )
   END_RUNG wire#w1
   // the same network as SCL:
   IF #TMR1.Q OR NOT #REDY THEN "DRV01-Bit_A" := TRUE; END_IF;
END_REGION

REGION Network 3: zalaczenie stycznika
   RUNG wire#powerrail
      Contact( #SUPV )
      Contact( "DRV01-Bit_A/M" )
      wire#w1
      Contact( "DRV01-Bit_REM" )
      I_Contact( "DRV01-Bit_A" )
      Coil( #CB )
   END_RUNG
   RUNG wire#powerrail
      Contact( "DRV01-Bit_Z" )
      wire#w2
      I_Contact( "DRV01-Bit_W" )
      I_Contact( "DRV01-Bit_A/M" )
   END_RUNG wire#w1
   RUNG wire#powerrail
      Contact( #RUN )
   END_RUNG wire#w2
   // the same network as SCL:
   #CB := ((#SUPV AND "DRV01-Bit_A/M") OR (("DRV01-Bit_Z" OR #RUN) AND NOT "DRV01-Bit_W" AND NOT "DRV01-Bit_A/M")) AND "DRV01-Bit_REM" AND NOT "DRV01-Bit_A";
END_REGION

REGION Network 4: Kontrola czasu na załączenie stycznika
   #TMR1(IN := ((#CB AND NOT #RUN) OR (NOT #CB AND #RUN)) AND "DRV01-Bit_REM", PT := #KT1);   // TON coil
END_REGION

REGION Network 5: Kasowanie DRV01-Bit_Awaria
   RUNG wire#powerrail
      Contact( "DRV01-Bit_R" )
      R_Coil( "DRV01-Bit_A" )
   END_RUNG
   // the same network as SCL:
   IF "DRV01-Bit_R" THEN "DRV01-Bit_A" := FALSE; END_IF;
END_REGION

REGION Network 6: Bit Out wektora napędu sygnał Alarm
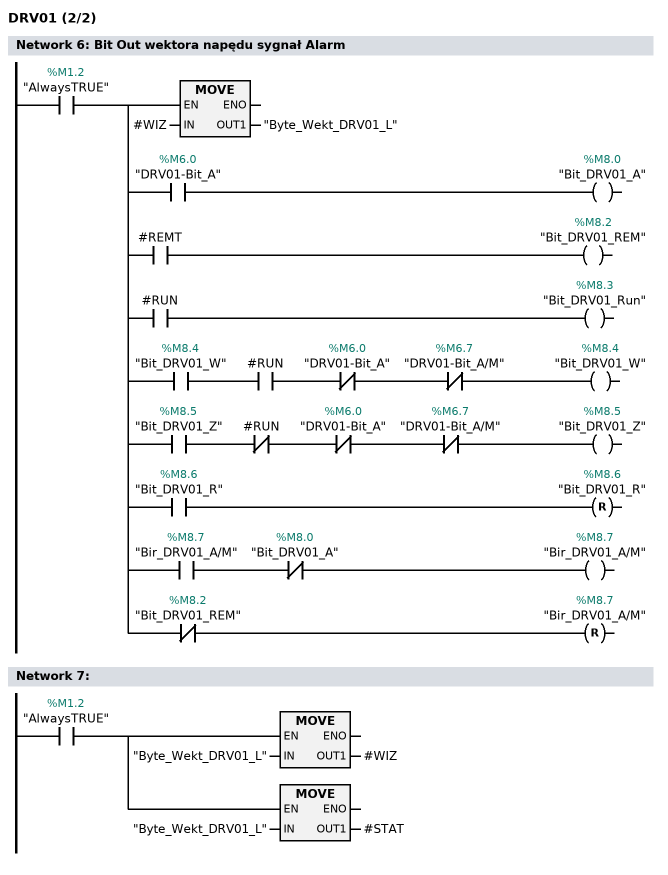
   RUNG wire#powerrail
      Contact( "AlwaysTRUE" )
      wire#w1
      { S7_GenerateENO := "TRUE" } Move(in := #WIZ, out1 => "Byte_Wekt_DRV01_L")
   END_RUNG
   RUNG wire#w1
      Contact( "DRV01-Bit_A" )
      Coil( "Bit_DRV01_A" )
   END_RUNG
   RUNG wire#w1
      Contact( #REMT )
      Coil( "Bit_DRV01_REM" )
   END_RUNG
   RUNG wire#w1
      Contact( #RUN )
      Coil( "Bit_DRV01_Run" )
   END_RUNG
   RUNG wire#w1
      Contact( "Bit_DRV01_W" )
      Contact( #RUN )
      I_Contact( "DRV01-Bit_A" )
      I_Contact( "DRV01-Bit_A/M" )
      Coil( "Bit_DRV01_W" )
   END_RUNG
   RUNG wire#w1
      Contact( "Bit_DRV01_Z" )
      I_Contact( #RUN )
      I_Contact( "DRV01-Bit_A" )
      I_Contact( "DRV01-Bit_A/M" )
      Coil( "Bit_DRV01_Z" )
   END_RUNG
   RUNG wire#w1
      Contact( "Bit_DRV01_R" )
      R_Coil( "Bit_DRV01_R" )
   END_RUNG
   RUNG wire#w1
      Contact( "Bir_DRV01_A/M" )
      I_Contact( "Bit_DRV01_A" )
      Coil( "Bir_DRV01_A/M" )
   END_RUNG
   RUNG wire#w1
      I_Contact( "Bit_DRV01_REM" )
      R_Coil( "Bir_DRV01_A/M" )
   END_RUNG
   // the same network as SCL:
   IF "AlwaysTRUE" THEN "Byte_Wekt_DRV01_L" := #WIZ; END_IF;
   "Bit_DRV01_A" := "AlwaysTRUE" AND "DRV01-Bit_A";
   "Bit_DRV01_REM" := "AlwaysTRUE" AND #REMT;
   "Bit_DRV01_Run" := "AlwaysTRUE" AND #RUN;
   "Bit_DRV01_W" := "AlwaysTRUE" AND "Bit_DRV01_W" AND #RUN AND NOT "DRV01-Bit_A" AND NOT "DRV01-Bit_A/M";
   "Bit_DRV01_Z" := "AlwaysTRUE" AND "Bit_DRV01_Z" AND NOT #RUN AND NOT "DRV01-Bit_A" AND NOT "DRV01-Bit_A/M";
   IF "AlwaysTRUE" AND "Bit_DRV01_R" THEN "Bit_DRV01_R" := FALSE; END_IF;
   "Bir_DRV01_A/M" := "AlwaysTRUE" AND "Bir_DRV01_A/M" AND NOT "Bit_DRV01_A";
   IF "AlwaysTRUE" AND NOT "Bit_DRV01_REM" THEN "Bir_DRV01_A/M" := FALSE; END_IF;
END_REGION

REGION Network 7
   RUNG wire#powerrail
      Contact( "AlwaysTRUE" )
      wire#w1
      { S7_GenerateENO := "TRUE" } Move(in := "Byte_Wekt_DRV01_L", out1 => #WIZ)
   END_RUNG
   RUNG wire#w1
      { S7_GenerateENO := "TRUE" } Move(in := "Byte_Wekt_DRV01_L", out1 => #STAT)
   END_RUNG
   // the same network as SCL:
   IF "AlwaysTRUE" THEN
       #WIZ := "Byte_Wekt_DRV01_L";
       #STAT := "Byte_Wekt_DRV01_L";
   END_IF;
END_REGION
END_FUNCTION

FUNCTION "Reset" : Void   // FC7, LAD
TITLE = Reset PID
{ S7_Optimized_Access := 'TRUE' }
AUTHOR : RTecmer
VERSION : 0.1
// (*
// //=============================================================================
// //(JZWiK S.A Radosław Tecmer)
// //(c)Copyright (2021) All Rights Reserved
// //-----------------------------------------------------------------------------
// //Testowane z:   (system docelowy z  FW 4.4)
// //Pakiet inżynierski:   TIA Portal (V14 Sp1 Update 9)
// //Ograniczenia:  ( - )
// //Wymagania:  (minimalne S7-1200 CPU 1215C FW 4.2 .)
// //Funkcjonalnośc: (Reset błędu i ustawienie wartości domyślnych PID )
// //-----------------------------------------------------------------------------
// //Zmainy wprowadzone:
// //Wersja  Data       Osoba wprowadzająca zmiany - ekspert
// //01.00.00 17.11.2021 (Tecmer Radosław - twórca) Pieresza wersja 01.00.00
// //=============================================================================
// *)
// stored: AutoNumber true, IsIECCheckEnabled false, SetENOAutomatically false, UDAEnableTagReadback false
BEGIN
END_FUNCTION

FUNCTION "Convert_analogs" : Void   // FC14, LAD
TITLE = Funkcja konwertera analogów
{ S7_Optimized_Access := 'TRUE' }
AUTHOR : RTecmer
VERSION : 0.1
// "Switch_set_OverCurrentInverer" - Porzełączni wyboru źródła wartości parametrówą falownika  ( 0- wartość z Modbus RTU, 1- wartość zadana ręcznie) / Konwertowanie zmiennych procesowych
// stored: AutoNumber true, IsIECCheckEnabled false, SetENOAutomatically false, UDAEnableTagReadback false
   VAR_TEMP   // added for the SCL form of the ladder/FBD networks
      _w1 : Bool;
   END_VAR
BEGIN

REGION Network 1: Przepywomierz Q1 Pompownia
   // Pobrane z Modbus RTU
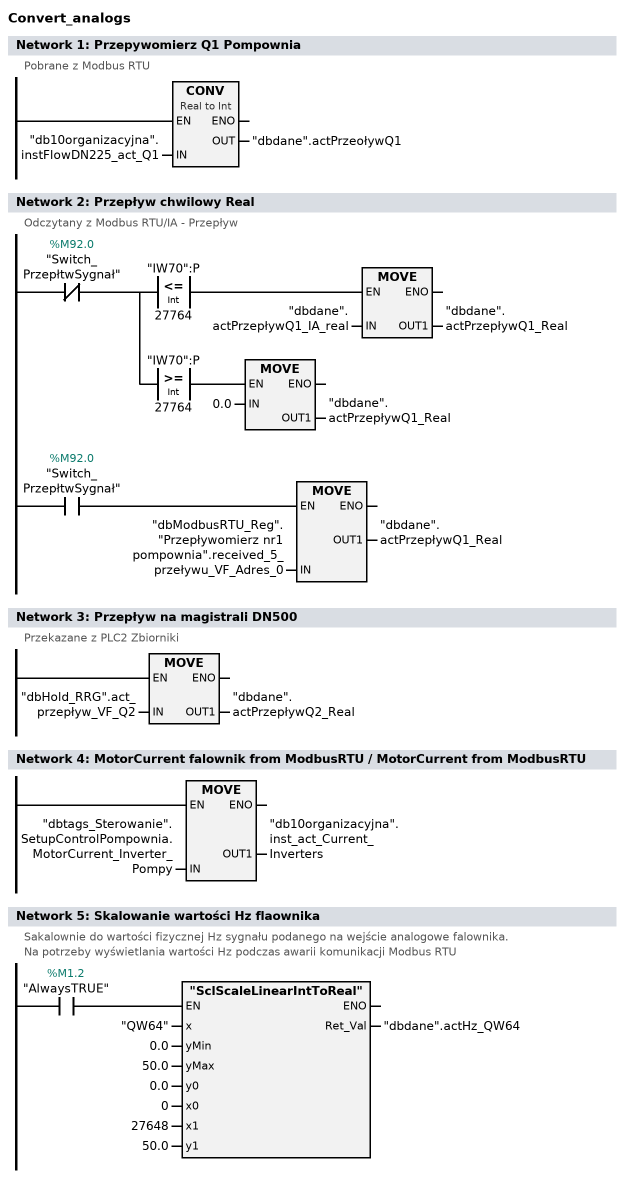
   RUNG wire#powerrail
      { S7_Templates := "[SrcType := Real, DestType := Int]" } Convert(in := "db10organizacyjna".instFlowDN225_act_Q1, out => "dbdane".actPrzeoływQ1)
   END_RUNG
   // the same network as SCL:
   "dbdane".actPrzeoływQ1 := REAL_TO_INT("db10organizacyjna".instFlowDN225_act_Q1);
END_REGION

REGION Network 2: Przepływ chwilowy Real
   // Odczytany z Modbus RTU/IA - Przepływ
   RUNG wire#powerrail
      I_Contact( "Switch_PrzepłtwSygnał" )
      wire#w1
      { S7_Templates := "SrcType := Int" } LE_Contact(in1 := "IW70":P, in2 := 27764)
      Move(in := "dbdane".actPrzepływQ1_IA_real, out1 => "dbdane".actPrzepływQ1_Real)
   END_RUNG
   RUNG wire#w1
      { S7_Templates := "SrcType := Int" } GE_Contact(in1 := "IW70":P, in2 := 27764)
      Move(in := 0.0, out1 => "dbdane".actPrzepływQ1_Real)
   END_RUNG
   RUNG wire#powerrail
      Contact( "Switch_PrzepłtwSygnał" )
      Move(in := "dbModbusRTU_Reg"."Przepływomierz nr1 pompownia".received_5_przeływu_VF_Adres_0, out1 => "dbdane".actPrzepływQ1_Real)
   END_RUNG
   // the same network as SCL:
   #_w1 := NOT "Switch_PrzepłtwSygnał";
   IF #_w1 AND ("IW70":P <= 27764) THEN
       "dbdane".actPrzepływQ1_Real := "dbdane".actPrzepływQ1_IA_real;
   END_IF;
   IF #_w1 AND ("IW70":P >= 27764) THEN "dbdane".actPrzepływQ1_Real := 0.0; END_IF;
   IF "Switch_PrzepłtwSygnał" THEN
       "dbdane".actPrzepływQ1_Real := "dbModbusRTU_Reg"."Przepływomierz nr1 pompownia".received_5_przeływu_VF_Adres_0;
   END_IF;
END_REGION

REGION Network 3: Przepływ na magistrali DN500
   // Przekazane z PLC2 Zbiorniki
   RUNG wire#powerrail
      Move(in := "dbHold_RRG".act_przepływ_VF_Q2, out1 => "dbdane".actPrzepływQ2_Real)
   END_RUNG
   // the same network as SCL:
   "dbdane".actPrzepływQ2_Real := "dbHold_RRG".act_przepływ_VF_Q2;
END_REGION

REGION Network 4: MotorCurrent falownik from ModbusRTU / MotorCurrent from ModbusRTU
   RUNG wire#powerrail
      Move(in := "dbtags_Sterowanie".SetupControlPompownia.MotorCurrent_Inverter_Pompy, out1 => "db10organizacyjna".inst_act_Current_Inverters)
   END_RUNG
   // the same network as SCL:
   "db10organizacyjna".inst_act_Current_Inverters := "dbtags_Sterowanie".SetupControlPompownia.MotorCurrent_Inverter_Pompy;
END_REGION

REGION Network 5: Skalowanie wartości Hz flaownika
   // Sakalownie do wartości fizycznej Hz sygnału podanego na wejście analogowe falownika.
   // Na potrzeby wyświetlania wartości Hz podczas awarii komunikacji Modbus RTU
   RUNG wire#powerrail
      Contact( "AlwaysTRUE" )
      "SclScaleLinearIntToReal"(x := "QW64", yMin := 0.0, yMax := 50.0, y0 := 0.0, x0 := 0, x1 := 27648, y1 := 50.0, Ret_Val => "dbdane".actHz_QW64)
   END_RUNG
   // the same network as SCL:
   IF "AlwaysTRUE" THEN
       "dbdane".actHz_QW64 := "SclScaleLinearIntToReal"(x := "QW64",
                               yMin := 0.0,
                               yMax := 50.0,
                               y0 := 0.0,
                               x0 := 0,
                               x1 := 27648,
                               y1 := 50.0);
   END_IF;
END_REGION
END_FUNCTION

FUNCTION "Obsługa alarmów" : Void   // FC10, LAD
TITLE = Boks Ready
{ S7_Optimized_Access := 'TRUE' }
AUTHOR : R.Tecmer
VERSION : 0.1
// Handling of alarms. Signaling and deleting
// stored: AutoNumber true, IsIECCheckEnabled false, SetENOAutomatically false, UDAEnableTagReadback false
BEGIN

REGION Network 1: Ready Inverters No1 No2
   // połączyłem bo usunięto drugi falownik
   // Jeśli brak gotowości to ustaw bity
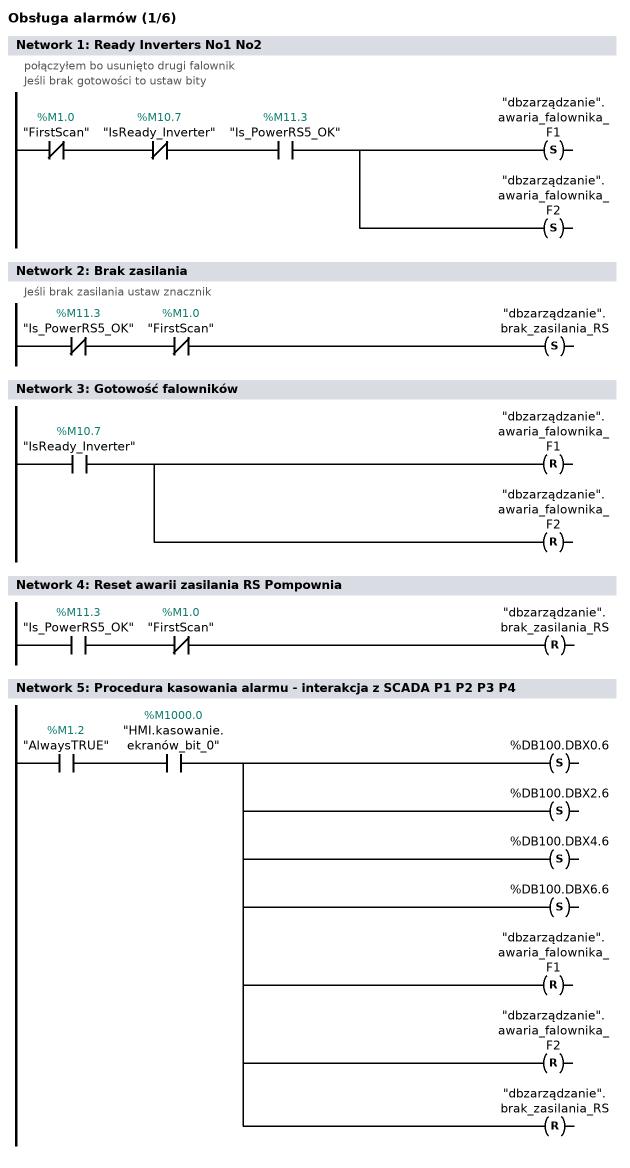
   RUNG wire#powerrail
      I_Contact( "FirstScan" )
      I_Contact( "IsReady_Inverter" )
      Contact( "Is_PowerRS5_OK" )
      wire#w1
      S_Coil( "dbzarządzanie".awaria_falownika_F1 )
   END_RUNG
   RUNG wire#w1
      S_Coil( "dbzarządzanie".awaria_falownika_F2 )
   END_RUNG
   // the same network as SCL:
   IF NOT "FirstScan" AND NOT "IsReady_Inverter" AND "Is_PowerRS5_OK" THEN
       "dbzarządzanie".awaria_falownika_F1 := TRUE;
       "dbzarządzanie".awaria_falownika_F2 := TRUE;
   END_IF;
END_REGION

REGION Network 2: Brak zasilania
   // Jeśli brak zasilania ustaw znacznik
   RUNG wire#powerrail
      I_Contact( "Is_PowerRS5_OK" )
      I_Contact( "FirstScan" )
      S_Coil( "dbzarządzanie".brak_zasilania_RS )
   END_RUNG
   // the same network as SCL:
   IF NOT "Is_PowerRS5_OK" AND NOT "FirstScan" THEN "dbzarządzanie".brak_zasilania_RS := TRUE; END_IF;
END_REGION

REGION Network 3: Gotowość falowników
   RUNG wire#powerrail
      Contact( "IsReady_Inverter" )
      wire#w1
      R_Coil( "dbzarządzanie".awaria_falownika_F1 )
   END_RUNG
   RUNG wire#w1
      R_Coil( "dbzarządzanie".awaria_falownika_F2 )
   END_RUNG
   // the same network as SCL:
   IF "IsReady_Inverter" THEN
       "dbzarządzanie".awaria_falownika_F1 := FALSE;
       "dbzarządzanie".awaria_falownika_F2 := FALSE;
   END_IF;
END_REGION

REGION Network 4: Reset awarii zasilania RS Pompownia
   RUNG wire#powerrail
      Contact( "Is_PowerRS5_OK" )
      I_Contact( "FirstScan" )
      R_Coil( "dbzarządzanie".brak_zasilania_RS )
   END_RUNG
   // the same network as SCL:
   IF "Is_PowerRS5_OK" AND NOT "FirstScan" THEN "dbzarządzanie".brak_zasilania_RS := FALSE; END_IF;
END_REGION

REGION Network 5: Procedura kasowania alarmu - interakcja z SCADA P1 P2 P3 P4
   RUNG wire#powerrail
      Contact( "AlwaysTRUE" )
      Contact( "HMI.kasowanie.ekranów_bit_0" )
      wire#w1
      S_Coil( %DB100.DBX0.6 )
   END_RUNG
   RUNG wire#w1
      S_Coil( %DB100.DBX2.6 )
   END_RUNG
   RUNG wire#w1
      S_Coil( %DB100.DBX4.6 )
   END_RUNG
   RUNG wire#w1
      S_Coil( %DB100.DBX6.6 )
   END_RUNG
   RUNG wire#w1
      R_Coil( "dbzarządzanie".awaria_falownika_F1 )
   END_RUNG
   RUNG wire#w1
      R_Coil( "dbzarządzanie".awaria_falownika_F2 )
   END_RUNG
   RUNG wire#w1
      R_Coil( "dbzarządzanie".brak_zasilania_RS )
   END_RUNG
   // the same network as SCL:
   IF "AlwaysTRUE" AND "HMI.kasowanie.ekranów_bit_0" THEN
       %DB100.DBX0.6 := TRUE;
       %DB100.DBX2.6 := TRUE;
       %DB100.DBX4.6 := TRUE;
       %DB100.DBX6.6 := TRUE;
       "dbzarządzanie".awaria_falownika_F1 := FALSE;
       "dbzarządzanie".awaria_falownika_F2 := FALSE;
       "dbzarządzanie".brak_zasilania_RS := FALSE;
   END_IF;
END_REGION

REGION Network 6: Reset błędu Soft-Start
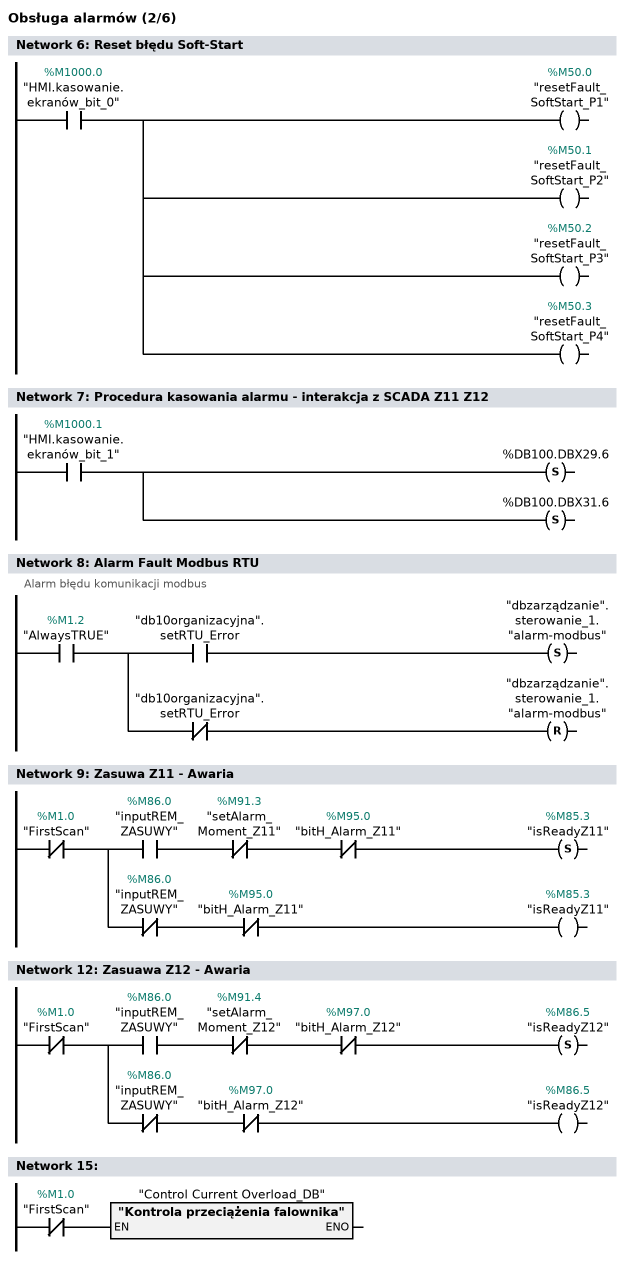
   RUNG wire#powerrail
      Contact( "HMI.kasowanie.ekranów_bit_0" )
      wire#w1
      Coil( "resetFault_SoftStart_P1" )
   END_RUNG
   RUNG wire#w1
      Coil( "resetFault_SoftStart_P2" )
   END_RUNG
   RUNG wire#w1
      Coil( "resetFault_SoftStart_P3" )
   END_RUNG
   RUNG wire#w1
      Coil( "resetFault_SoftStart_P4" )
   END_RUNG
   // the same network as SCL:
   "resetFault_SoftStart_P1" := "HMI.kasowanie.ekranów_bit_0";
   "resetFault_SoftStart_P2" := "HMI.kasowanie.ekranów_bit_0";
   "resetFault_SoftStart_P3" := "HMI.kasowanie.ekranów_bit_0";
   "resetFault_SoftStart_P4" := "HMI.kasowanie.ekranów_bit_0";
END_REGION

REGION Network 7: Procedura kasowania alarmu - interakcja z SCADA Z11 Z12
   RUNG wire#powerrail
      Contact( "HMI.kasowanie.ekranów_bit_1" )
      wire#w1
      S_Coil( %DB100.DBX29.6 )
   END_RUNG
   RUNG wire#w1
      S_Coil( %DB100.DBX31.6 )
   END_RUNG
   // the same network as SCL:
   IF "HMI.kasowanie.ekranów_bit_1" THEN
       %DB100.DBX29.6 := TRUE;
       %DB100.DBX31.6 := TRUE;
   END_IF;
END_REGION

REGION Network 8: Alarm Fault Modbus RTU
   // Alarm błędu komunikacji modbus
   RUNG wire#powerrail
      Contact( "AlwaysTRUE" )
      wire#w1
      Contact( "db10organizacyjna".setRTU_Error )
      S_Coil( "dbzarządzanie".sterowanie_1."alarm-modbus" )
   END_RUNG
   RUNG wire#w1
      I_Contact( "db10organizacyjna".setRTU_Error )
      R_Coil( "dbzarządzanie".sterowanie_1."alarm-modbus" )
   END_RUNG
   // the same network as SCL:
   IF "AlwaysTRUE" AND "db10organizacyjna".setRTU_Error THEN
       "dbzarządzanie".sterowanie_1."alarm-modbus" := TRUE;
   END_IF;
   IF "AlwaysTRUE" AND NOT "db10organizacyjna".setRTU_Error THEN
       "dbzarządzanie".sterowanie_1."alarm-modbus" := FALSE;
   END_IF;
END_REGION

REGION Network 9: Zasuwa Z11 - Awaria
   RUNG wire#powerrail
      I_Contact( "FirstScan" )
      wire#w1
      Contact( "inputREM_ZASUWY" )
      I_Contact( "setAlarm_Moment_Z11" )
      I_Contact( "bitH_Alarm_Z11" )
      S_Coil( "isReadyZ11" )
   END_RUNG
   RUNG wire#w1
      I_Contact( "inputREM_ZASUWY" )
      I_Contact( "bitH_Alarm_Z11" )
      Coil( "isReadyZ11" )
   END_RUNG
   // the same network as SCL:
   IF NOT "FirstScan" AND "inputREM_ZASUWY" AND NOT "setAlarm_Moment_Z11" AND NOT "bitH_Alarm_Z11" THEN
       "isReadyZ11" := TRUE;
   END_IF;
   "isReadyZ11" := NOT "FirstScan" AND NOT "inputREM_ZASUWY" AND NOT "bitH_Alarm_Z11";
END_REGION

REGION Network 10 (SCL): Z11 znacznik alarmu od momentówki w trybie zdalnym (aut/mamnual)
   IF  "inputAwariaMomentZ11" = False THEN
     // Ustaw alarm od momentu
     "setAlarm_Moment_Z11" := TRUE;
   ELSE
     "setAlarm_Moment_Z11" := FALSE;
     ;
   END_IF;
END_REGION

REGION Network 11 (SCL): Ustaw brak gotowości Z11
   IF "setAlarm_Moment_Z11" = TRUE OR "bitH_Alarm_Z11" THEN
     // Ustaw Alarm
     "isReadyZ11" := FALSE;

     ;
   END_IF;
END_REGION

REGION Network 12: Zasuawa Z12 - Awaria
   RUNG wire#powerrail
      I_Contact( "FirstScan" )
      wire#w1
      Contact( "inputREM_ZASUWY" )
      I_Contact( "setAlarm_Moment_Z12" )
      I_Contact( "bitH_Alarm_Z12" )
      S_Coil( "isReadyZ12" )
   END_RUNG
   RUNG wire#w1
      I_Contact( "inputREM_ZASUWY" )
      I_Contact( "bitH_Alarm_Z12" )
      Coil( "isReadyZ12" )
   END_RUNG
   // the same network as SCL:
   IF NOT "FirstScan" AND "inputREM_ZASUWY" AND NOT "setAlarm_Moment_Z12" AND NOT "bitH_Alarm_Z12" THEN
       "isReadyZ12" := TRUE;
   END_IF;
   "isReadyZ12" := NOT "FirstScan" AND NOT "inputREM_ZASUWY" AND NOT "bitH_Alarm_Z12";
END_REGION

REGION Network 13 (SCL): Z12 znacznik alarmu od momentówki w trybie zdalnym (aut/mamnual)
   IF "inputAwariaMomentZ12" = False THEN
     // Ustaw alarm od momentu
     "setAlarm_Moment_Z12" := TRUE;
   ELSE
     "setAlarm_Moment_Z12" := FALSE;
     ;
   END_IF;
END_REGION

REGION Network 14 (SCL): Ustaw brak gotowości Z12
   IF "setAlarm_Moment_Z12" = TRUE OR "bitH_Alarm_Z12" THEN
     // Ustaw Alarm
     "isReadyZ12" := FALSE;

     ;
   END_IF;
END_REGION

REGION Network 15
   RUNG wire#powerrail
      I_Contact( "FirstScan" )
      "Control Current Overload_DB"()
   END_RUNG
   // the same network as SCL:
   IF NOT "FirstScan" THEN
       "Control Current Overload_DB"();   // "Kontrola przeciążenia falownika"
   END_IF;
END_REGION

REGION Network 16: Controla ciśnienia na rurociągu tłoczenia
   // Ciśnienie mierzone w kierunku tłoczenia
   // Jeśli max ustaw alarm
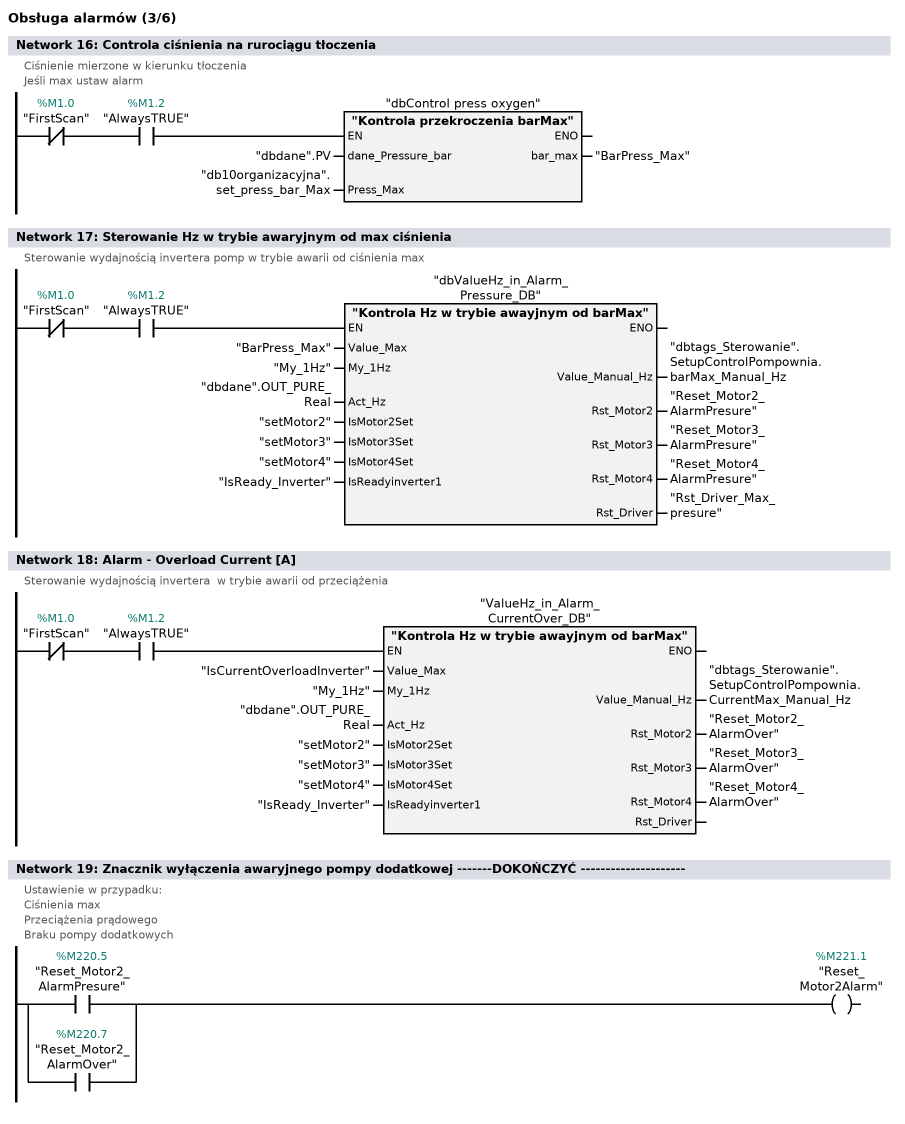
   RUNG wire#powerrail
      I_Contact( "FirstScan" )
      Contact( "AlwaysTRUE" )
      "dbControl press oxygen"(dane_Pressure_bar := "dbdane".PV, Press_Max := "db10organizacyjna".set_press_bar_Max, bar_max => "BarPress_Max")
   END_RUNG
   // the same network as SCL:
   IF NOT "FirstScan" AND "AlwaysTRUE" THEN
       "dbControl press oxygen"(dane_Pressure_bar := "dbdane".PV,   // "Kontrola przekroczenia barMax"
                               Press_Max := "db10organizacyjna".set_press_bar_Max,
                               bar_max => "BarPress_Max");
   END_IF;
END_REGION

REGION Network 17: Sterowanie Hz w trybie awaryjnym od max ciśnienia
   // Sterowanie wydajnością invertera pomp w trybie awarii od ciśnienia max
   RUNG wire#powerrail
      I_Contact( "FirstScan" )
      Contact( "AlwaysTRUE" )
      "dbValueHz_in_Alarm_Pressure_DB"(Value_Max := "BarPress_Max", My_1Hz := "My_1Hz", Act_Hz := "dbdane".OUT_PURE_Real, IsMotor2Set := "setMotor2", IsMotor3Set := "setMotor3", IsMotor4Set := "setMotor4", IsReadyinverter1 := "IsReady_Inverter", Value_Manual_Hz => "dbtags_Sterowanie".SetupControlPompownia.barMax_Manual_Hz, Rst_Motor2 => "Reset_Motor2_AlarmPresure", Rst_Motor3 => "Reset_Motor3_AlarmPresure", Rst_Motor4 => "Reset_Motor4_AlarmPresure", Rst_Driver => "Rst_Driver_Max_presure")
   END_RUNG
   // the same network as SCL:
   IF NOT "FirstScan" AND "AlwaysTRUE" THEN
       "dbValueHz_in_Alarm_Pressure_DB"(Value_Max := "BarPress_Max",   // "Kontrola Hz w trybie awayjnym od barMax"
                               My_1Hz := "My_1Hz",
                               Act_Hz := "dbdane".OUT_PURE_Real,
                               IsMotor2Set := "setMotor2",
                               IsMotor3Set := "setMotor3",
                               IsMotor4Set := "setMotor4",
                               IsReadyinverter1 := "IsReady_Inverter",
                               Value_Manual_Hz => "dbtags_Sterowanie".SetupControlPompownia.barMax_Manual_Hz,
                               Rst_Motor2 => "Reset_Motor2_AlarmPresure",
                               Rst_Motor3 => "Reset_Motor3_AlarmPresure",
                               Rst_Motor4 => "Reset_Motor4_AlarmPresure",
                               Rst_Driver => "Rst_Driver_Max_presure");
   END_IF;
END_REGION

REGION Network 18: Alarm - Overload Current [A]
   // Sterowanie wydajnością invertera  w trybie awarii od przeciążenia
   RUNG wire#powerrail
      I_Contact( "FirstScan" )
      Contact( "AlwaysTRUE" )
      "ValueHz_in_Alarm_CurrentOver_DB"(Value_Max := "IsCurrentOverloadInverter", My_1Hz := "My_1Hz", Act_Hz := "dbdane".OUT_PURE_Real, IsMotor2Set := "setMotor2", IsMotor3Set := "setMotor3", IsMotor4Set := "setMotor4", IsReadyinverter1 := "IsReady_Inverter", Value_Manual_Hz => "dbtags_Sterowanie".SetupControlPompownia.CurrentMax_Manual_Hz, Rst_Motor2 => "Reset_Motor2_AlarmOver", Rst_Motor3 => "Reset_Motor3_AlarmOver", Rst_Motor4 => "Reset_Motor4_AlarmOver", Rst_Driver =>)
   END_RUNG
   // the same network as SCL:
   IF NOT "FirstScan" AND "AlwaysTRUE" THEN
       "ValueHz_in_Alarm_CurrentOver_DB"(Value_Max := "IsCurrentOverloadInverter",   // "Kontrola Hz w trybie awayjnym od barMax"
                               My_1Hz := "My_1Hz",
                               Act_Hz := "dbdane".OUT_PURE_Real,
                               IsMotor2Set := "setMotor2",
                               IsMotor3Set := "setMotor3",
                               IsMotor4Set := "setMotor4",
                               IsReadyinverter1 := "IsReady_Inverter",
                               Value_Manual_Hz => "dbtags_Sterowanie".SetupControlPompownia.CurrentMax_Manual_Hz,
                               Rst_Motor2 => "Reset_Motor2_AlarmOver",
                               Rst_Motor3 => "Reset_Motor3_AlarmOver",
                               Rst_Motor4 => "Reset_Motor4_AlarmOver");
   END_IF;
END_REGION

REGION Network 19: Znacznik wyłączenia awaryjnego pompy dodatkowej -------DOKOŃCZYĆ ---------------------
   // Ustawienie w przypadku:
   // Ciśnienia max
   // Przeciążenia prądowego
   // Braku pompy dodatkowych
   RUNG wire#powerrail
      Contact( "Reset_Motor2_AlarmPresure" )
      wire#w1
      Coil( "Reset_Motor2Alarm" )
   END_RUNG
   RUNG wire#powerrail
      Contact( "Reset_Motor2_AlarmOver" )
   END_RUNG wire#w1
   // the same network as SCL:
   "Reset_Motor2Alarm" := "Reset_Motor2_AlarmPresure" OR "Reset_Motor2_AlarmOver";
END_REGION

REGION Network 20: Znacznik wyłączenia awaryjnego pompy dodatkowej
   // Ustawienie w przypadku:
   // Ciśnienia max
   // Przeciążenia prądowego
   // Braku pompy dodatkowych
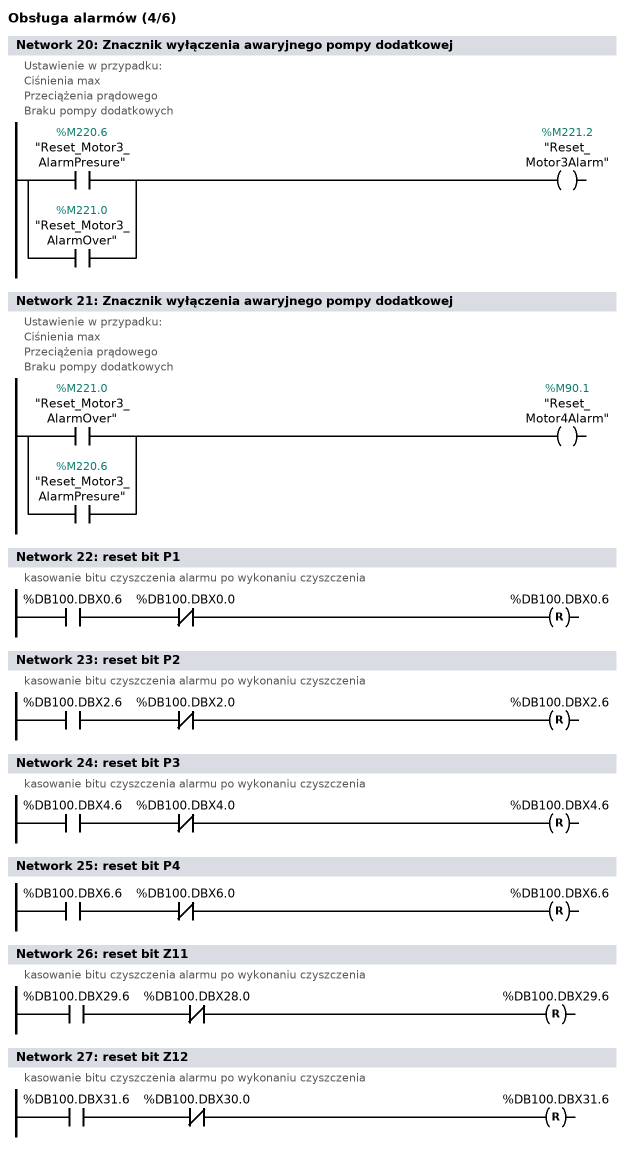
   RUNG wire#powerrail
      Contact( "Reset_Motor3_AlarmPresure" )
      wire#w1
      Coil( "Reset_Motor3Alarm" )
   END_RUNG
   RUNG wire#powerrail
      Contact( "Reset_Motor3_AlarmOver" )
   END_RUNG wire#w1
   // the same network as SCL:
   "Reset_Motor3Alarm" := "Reset_Motor3_AlarmPresure" OR "Reset_Motor3_AlarmOver";
END_REGION

REGION Network 21: Znacznik wyłączenia awaryjnego pompy dodatkowej
   // Ustawienie w przypadku:
   // Ciśnienia max
   // Przeciążenia prądowego
   // Braku pompy dodatkowych
   RUNG wire#powerrail
      Contact( "Reset_Motor3_AlarmOver" )
      wire#w1
      Coil( "Reset_Motor4Alarm" )
   END_RUNG
   RUNG wire#powerrail
      Contact( "Reset_Motor3_AlarmPresure" )
   END_RUNG wire#w1
   // the same network as SCL:
   "Reset_Motor4Alarm" := "Reset_Motor3_AlarmOver" OR "Reset_Motor3_AlarmPresure";
END_REGION

REGION Network 22: reset bit P1
   // kasowanie bitu czyszczenia alarmu po wykonaniu czyszczenia
   RUNG wire#powerrail
      Contact( %DB100.DBX0.6 )
      I_Contact( %DB100.DBX0.0 )
      R_Coil( %DB100.DBX0.6 )
   END_RUNG
   // the same network as SCL:
   IF %DB100.DBX0.6 AND NOT %DB100.DBX0.0 THEN %DB100.DBX0.6 := FALSE; END_IF;
END_REGION

REGION Network 23: reset bit P2
   // kasowanie bitu czyszczenia alarmu po wykonaniu czyszczenia
   RUNG wire#powerrail
      Contact( %DB100.DBX2.6 )
      I_Contact( %DB100.DBX2.0 )
      R_Coil( %DB100.DBX2.6 )
   END_RUNG
   // the same network as SCL:
   IF %DB100.DBX2.6 AND NOT %DB100.DBX2.0 THEN %DB100.DBX2.6 := FALSE; END_IF;
END_REGION

REGION Network 24: reset bit P3
   // kasowanie bitu czyszczenia alarmu po wykonaniu czyszczenia
   RUNG wire#powerrail
      Contact( %DB100.DBX4.6 )
      I_Contact( %DB100.DBX4.0 )
      R_Coil( %DB100.DBX4.6 )
   END_RUNG
   // the same network as SCL:
   IF %DB100.DBX4.6 AND NOT %DB100.DBX4.0 THEN %DB100.DBX4.6 := FALSE; END_IF;
END_REGION

REGION Network 25: reset bit P4
   RUNG wire#powerrail
      Contact( %DB100.DBX6.6 )
      I_Contact( %DB100.DBX6.0 )
      R_Coil( %DB100.DBX6.6 )
   END_RUNG
   // the same network as SCL:
   IF %DB100.DBX6.6 AND NOT %DB100.DBX6.0 THEN %DB100.DBX6.6 := FALSE; END_IF;
END_REGION

REGION Network 26: reset bit Z11
   // kasowanie bitu czyszczenia alarmu po wykonaniu czyszczenia
   RUNG wire#powerrail
      Contact( %DB100.DBX29.6 )
      I_Contact( %DB100.DBX28.0 )
      R_Coil( %DB100.DBX29.6 )
   END_RUNG
   // the same network as SCL:
   IF %DB100.DBX29.6 AND NOT %DB100.DBX28.0 THEN %DB100.DBX29.6 := FALSE; END_IF;
END_REGION

REGION Network 27: reset bit Z12
   // kasowanie bitu czyszczenia alarmu po wykonaniu czyszczenia
   RUNG wire#powerrail
      Contact( %DB100.DBX31.6 )
      I_Contact( %DB100.DBX30.0 )
      R_Coil( %DB100.DBX31.6 )
   END_RUNG
   // the same network as SCL:
   IF %DB100.DBX31.6 AND NOT %DB100.DBX30.0 THEN %DB100.DBX31.6 := FALSE; END_IF;
END_REGION

REGION Network 28: Reset Bitu Kasowania Alarmów
   // Po wykonaniu kasowania alarmów bit -0 jest zerowany
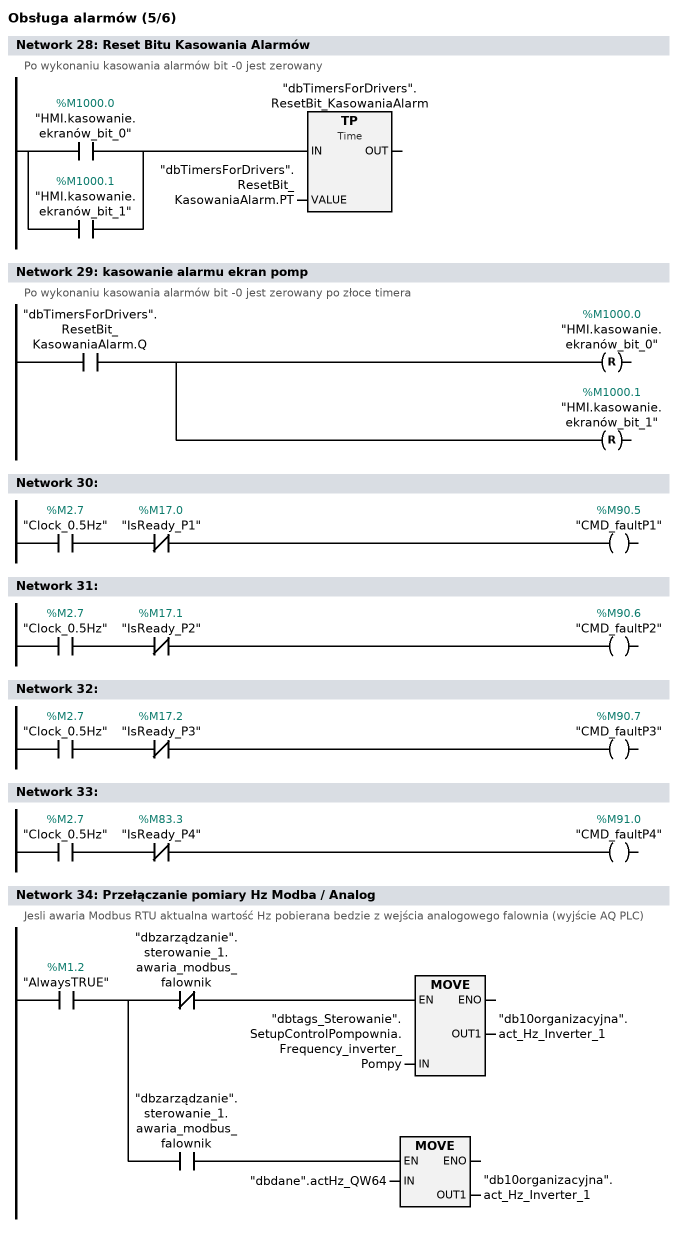
   "dbTimersForDrivers".ResetBit_KasowaniaAlarm.TP(IN := "HMI.kasowanie.ekranów_bit_0" OR "HMI.kasowanie.ekranów_bit_1", PT := "dbTimersForDrivers".ResetBit_KasowaniaAlarm.PT);   // TP coil
END_REGION

REGION Network 29: kasowanie alarmu ekran pomp
   // Po wykonaniu kasowania alarmów bit -0 jest zerowany po złoce timera
   RUNG wire#powerrail
      Contact( "dbTimersForDrivers".ResetBit_KasowaniaAlarm.Q )
      wire#w1
      R_Coil( "HMI.kasowanie.ekranów_bit_0" )
   END_RUNG
   RUNG wire#w1
      R_Coil( "HMI.kasowanie.ekranów_bit_1" )
   END_RUNG
   // the same network as SCL:
   IF "dbTimersForDrivers".ResetBit_KasowaniaAlarm.Q THEN
       "HMI.kasowanie.ekranów_bit_0" := FALSE;
       "HMI.kasowanie.ekranów_bit_1" := FALSE;
   END_IF;
END_REGION

REGION Network 30
   RUNG wire#powerrail
      Contact( "Clock_0.5Hz" )
      I_Contact( "IsReady_P1" )
      Coil( "CMD_faultP1" )
   END_RUNG
   // the same network as SCL:
   "CMD_faultP1" := "Clock_0.5Hz" AND NOT "IsReady_P1";
END_REGION

REGION Network 31
   RUNG wire#powerrail
      Contact( "Clock_0.5Hz" )
      I_Contact( "IsReady_P2" )
      Coil( "CMD_faultP2" )
   END_RUNG
   // the same network as SCL:
   "CMD_faultP2" := "Clock_0.5Hz" AND NOT "IsReady_P2";
END_REGION

REGION Network 32
   RUNG wire#powerrail
      Contact( "Clock_0.5Hz" )
      I_Contact( "IsReady_P3" )
      Coil( "CMD_faultP3" )
   END_RUNG
   // the same network as SCL:
   "CMD_faultP3" := "Clock_0.5Hz" AND NOT "IsReady_P3";
END_REGION

REGION Network 33
   RUNG wire#powerrail
      Contact( "Clock_0.5Hz" )
      I_Contact( "IsReady_P4" )
      Coil( "CMD_faultP4" )
   END_RUNG
   // the same network as SCL:
   "CMD_faultP4" := "Clock_0.5Hz" AND NOT "IsReady_P4";
END_REGION

REGION Network 34: Przełączanie pomiary Hz Modba / Analog
   // Jesli awaria Modbus RTU aktualna wartość Hz pobierana bedzie z wejścia analogowego falownia (wyjście AQ PLC)
   RUNG wire#powerrail
      Contact( "AlwaysTRUE" )
      wire#w1
      I_Contact( "dbzarządzanie".sterowanie_1.awaria_modbus_falownik )
      Move(in := "dbtags_Sterowanie".SetupControlPompownia.Frequency_inverter_Pompy, out1 => "db10organizacyjna".act_Hz_Inverter_1)
   END_RUNG
   RUNG wire#w1
      Contact( "dbzarządzanie".sterowanie_1.awaria_modbus_falownik )
      Move(in := "dbdane".actHz_QW64, out1 => "db10organizacyjna".act_Hz_Inverter_1)
   END_RUNG
   // the same network as SCL:
   IF "AlwaysTRUE" AND NOT "dbzarządzanie".sterowanie_1.awaria_modbus_falownik THEN
       "db10organizacyjna".act_Hz_Inverter_1 := "dbtags_Sterowanie".SetupControlPompownia.Frequency_inverter_Pompy;
   END_IF;
   IF "AlwaysTRUE" AND "dbzarządzanie".sterowanie_1.awaria_modbus_falownik THEN
       "db10organizacyjna".act_Hz_Inverter_1 := "dbdane".actHz_QW64;
   END_IF;
END_REGION

REGION Network 35: Q1 przepływomierz pompownia
   // zerowanie przepływu chwilowego gdy błąd komunikacji modbus z przepływomierzem
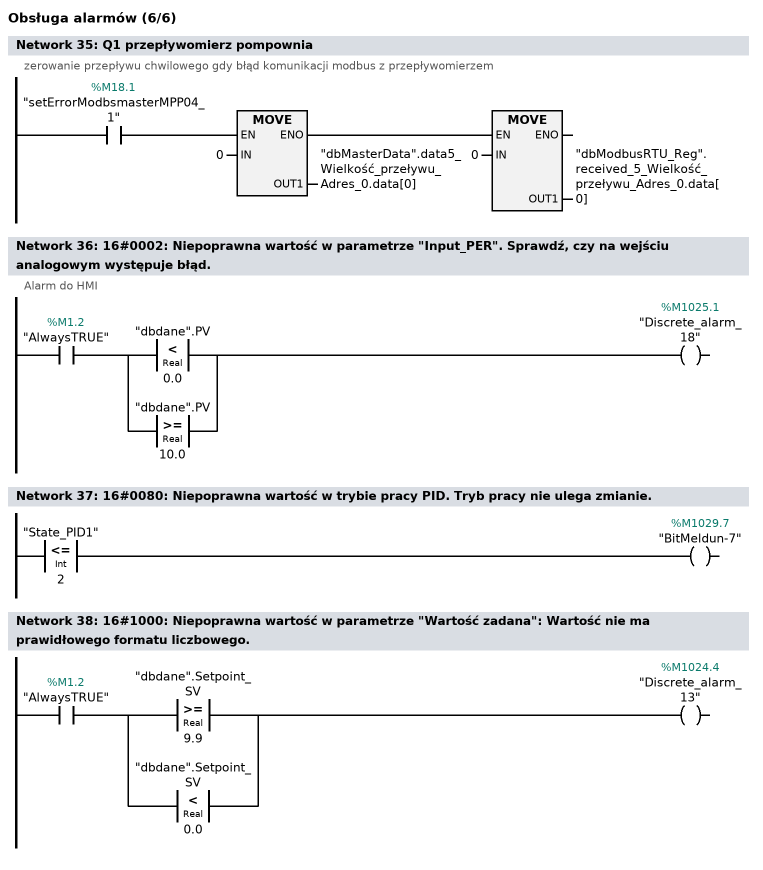
   RUNG wire#powerrail
      Contact( "setErrorModbsmasterMPP04_1" )
      { S7_GenerateENO := "TRUE" } Move(in := 0, out1 => "dbMasterData".data5_Wielkość_przeływu_Adres_0.data[0])
      { S7_GenerateENO := "TRUE" } Move(in := 0, out1 => "dbModbusRTU_Reg".received_5_Wielkość_przeływu_Adres_0.data[0])
   END_RUNG
   // the same network as SCL:
   // ENO of a box is taken as its EN; it also drops when the box reports an error
   IF "setErrorModbsmasterMPP04_1" THEN
       "dbMasterData".data5_Wielkość_przeływu_Adres_0.data[0] := 0;
       "dbModbusRTU_Reg".received_5_Wielkość_przeływu_Adres_0.data[0] := 0;
   END_IF;
END_REGION

REGION Network 36: 16#0002: Niepoprawna wartość w parametrze "Input_PER". Sprawdź, czy na wejściu analogowym występuje błąd.
   // Alarm do HMI
   RUNG wire#powerrail
      Contact( "AlwaysTRUE" )
      wire#w1
      { S7_Templates := "SrcType := Real" } LT_Contact(in1 := "dbdane".PV, in2 := 0.0)
      wire#w2
      Coil( "Discrete_alarm_18" )
   END_RUNG
   RUNG wire#w1
      { S7_Templates := "SrcType := Real" } GE_Contact(in1 := "dbdane".PV, in2 := 10.0)
   END_RUNG wire#w2
   // the same network as SCL:
   "Discrete_alarm_18" := "AlwaysTRUE" AND (("dbdane".PV < 0.0) OR ("dbdane".PV >= 10.0));
END_REGION

REGION Network 37: 16#0080: Niepoprawna wartość w trybie pracy PID. Tryb pracy nie ulega zmianie.
   RUNG wire#powerrail
      { S7_Templates := "SrcType := Int" } LE_Contact(in1 := "State_PID1", in2 := 2)
      Coil( "BitMeldun-7" )
   END_RUNG
   // the same network as SCL:
   "BitMeldun-7" := "State_PID1" <= 2;
END_REGION

REGION Network 38: 16#1000: Niepoprawna wartość w parametrze "Wartość zadana": Wartość nie ma prawidłowego formatu liczbowego.
   RUNG wire#powerrail
      Contact( "AlwaysTRUE" )
      wire#w1
      { S7_Templates := "SrcType := Real" } GE_Contact(in1 := "dbdane".Setpoint_SV, in2 := 9.9)
      wire#w2
      Coil( "Discrete_alarm_13" )
   END_RUNG
   RUNG wire#w1
      { S7_Templates := "SrcType := Real" } LT_Contact(in1 := "dbdane".Setpoint_SV, in2 := 0.0)
   END_RUNG wire#w2
   // the same network as SCL:
   "Discrete_alarm_13" := "AlwaysTRUE" AND (("dbdane".Setpoint_SV >= 9.9) OR ("dbdane".Setpoint_SV < 0.0));
END_REGION
END_FUNCTION

FUNCTION_BLOCK "Kontrola przeciążenia falownika"   // FB17, LAD
TITLE = Control Current Overload
{ S7_Optimized_Access := 'TRUE' }
AUTHOR : rtecmer
VERSION : 0.1
// Kontrola przeciążenia invertera KDN M25 M27
// stored: AutoNumber true, IsIECCheckEnabled false, IsRetainMemResEnabled false, MemoryReserve 500, SetENOAutomatically false, UDAEnableTagReadback false
BEGIN

REGION Network 1: Ustawienie wartości granicznej
   // Nastawa dopuszczalnego prądu invertera. Znacznik M10 zastosowany w celach serwisowych. Wybór ograniczenia z edytowanego z HMI lub z nastaw czytanych z falownika.
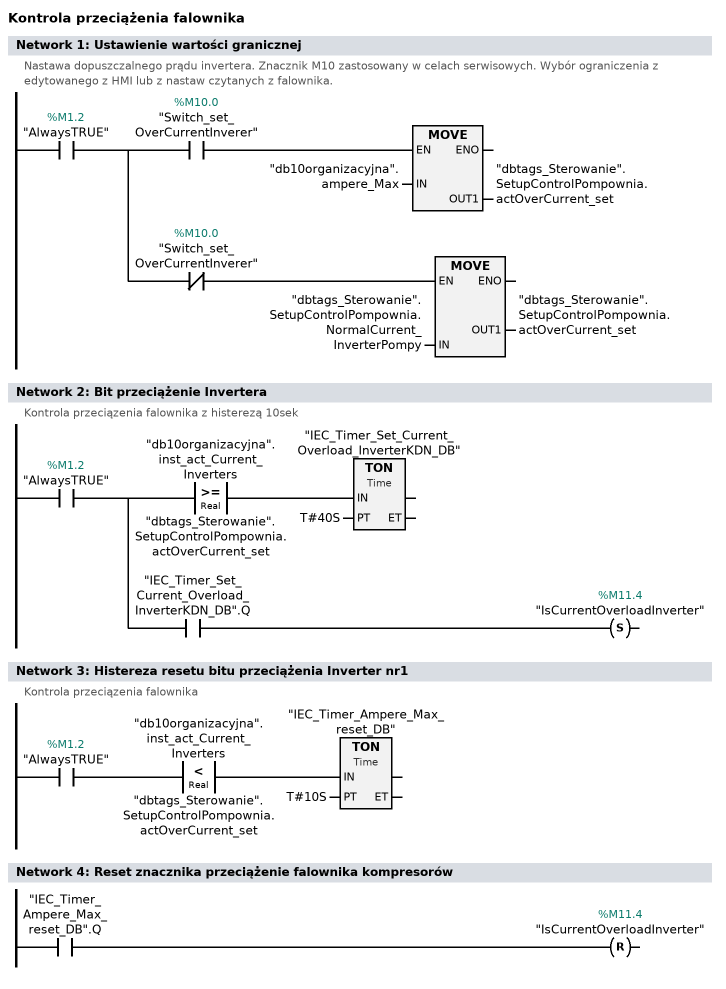
   RUNG wire#powerrail
      Contact( "AlwaysTRUE" )
      wire#w1
      Contact( "Switch_set_OverCurrentInverer" )
      Move(in := "db10organizacyjna".ampere_Max, out1 => "dbtags_Sterowanie".SetupControlPompownia.actOverCurrent_set)
   END_RUNG
   RUNG wire#w1
      I_Contact( "Switch_set_OverCurrentInverer" )
      Move(in := "dbtags_Sterowanie".SetupControlPompownia.NormalCurrent_InverterPompy, out1 => "dbtags_Sterowanie".SetupControlPompownia.actOverCurrent_set)
   END_RUNG
   // the same network as SCL:
   IF "AlwaysTRUE" AND "Switch_set_OverCurrentInverer" THEN
       "dbtags_Sterowanie".SetupControlPompownia.actOverCurrent_set := "db10organizacyjna".ampere_Max;
   END_IF;
   IF "AlwaysTRUE" AND NOT "Switch_set_OverCurrentInverer" THEN
       "dbtags_Sterowanie".SetupControlPompownia.actOverCurrent_set := "dbtags_Sterowanie".SetupControlPompownia.NormalCurrent_InverterPompy;
   END_IF;
END_REGION

REGION Network 2: Bit przeciążenie Invertera
   // Kontrola przeciązenia falownika z histerezą 10sek
   RUNG wire#powerrail
      Contact( "AlwaysTRUE" )
      wire#w1
      { S7_Templates := "SrcType := Real" } GE_Contact(in1 := "db10organizacyjna".inst_act_Current_Inverters, in2 := "dbtags_Sterowanie".SetupControlPompownia.actOverCurrent_set)
      { S7_Templates := "time_type := Time" } "IEC_Timer_Set_Current_Overload_InverterKDN_DB".TON(pt := T#40S, et =>)
   END_RUNG
   RUNG wire#w1
      Contact( "IEC_Timer_Set_Current_Overload_InverterKDN_DB".Q )
      S_Coil( "IsCurrentOverloadInverter" )
   END_RUNG
   // the same network as SCL:
   "IEC_Timer_Set_Current_Overload_InverterKDN_DB".TON(IN := "AlwaysTRUE" AND ("db10organizacyjna".inst_act_Current_Inverters >= "dbtags_Sterowanie".SetupControlPompownia.actOverCurrent_set),
                           PT := T#40S);
   IF "AlwaysTRUE" AND "IEC_Timer_Set_Current_Overload_InverterKDN_DB".Q THEN
       "IsCurrentOverloadInverter" := TRUE;
   END_IF;
END_REGION

REGION Network 3: Histereza resetu bitu przeciążenia Inverter nr1
   // Kontrola przeciązenia falownika
   RUNG wire#powerrail
      Contact( "AlwaysTRUE" )
      { S7_Templates := "SrcType := Real" } LT_Contact(in1 := "db10organizacyjna".inst_act_Current_Inverters, in2 := "dbtags_Sterowanie".SetupControlPompownia.actOverCurrent_set)
      { S7_Templates := "time_type := Time" } "IEC_Timer_Ampere_Max_reset_DB".TON(pt := T#10S, et =>)
   END_RUNG
   // the same network as SCL:
   "IEC_Timer_Ampere_Max_reset_DB".TON(IN := "AlwaysTRUE" AND ("db10organizacyjna".inst_act_Current_Inverters < "dbtags_Sterowanie".SetupControlPompownia.actOverCurrent_set),
                           PT := T#10S);
END_REGION

REGION Network 4: Reset znacznika przeciążenie falownika kompresorów
   RUNG wire#powerrail
      Contact( "IEC_Timer_Ampere_Max_reset_DB".Q )
      R_Coil( "IsCurrentOverloadInverter" )
   END_RUNG
   // the same network as SCL:
   IF "IEC_Timer_Ampere_Max_reset_DB".Q THEN "IsCurrentOverloadInverter" := FALSE; END_IF;
END_REGION
END_FUNCTION_BLOCK

FUNCTION_BLOCK "Kontrola przekroczenia barMax"
TITLE = Control press oxygen 
{ S7_Optimized_Access := 'TRUE' }
AUTHOR : rtecmer
VERSION : 0.1
//KOntrola ciśnienia w rurociągu. Sterowanie ograniczeniem wydajności falownika w przypadku przekroczenia ciśnienia max
   VAR_INPUT 
      dane_Pressure_bar : Real;   // Aktualne ciśnienie w rurociągu
      Press_Max { ExternalAccessible := 'False'; ExternalVisible := 'False'; ExternalWritable := 'False'} : Real;   // Ciśnienie graniczne max
   END_VAR

   VAR_OUTPUT 
      bar_max : Bool;   // Bit sygnału alarm ciśnienie za wysokie w rurociągu
   END_VAR

   VAR_TEMP 
      Temp_Press_max : Bool;   // Znacznik pomocniczy
   END_VAR


BEGIN
	//Kontrola cieśnienia granicznego w rurociągu 
	//
	
	REGION Control Press
	  // Porównanie aktualnego z Max
	  IF #dane_Pressure_bar > #Press_Max THEN
	    // Ustawienie znacznika jeśli Act > Max
	    #Temp_Press_max := TRUE;
	  ELSE
	    #Temp_Press_max := FALSE;
	    ;
	  END_IF;
	  
	 "IEC_Timer_PressO2_Max_DB".TON(IN:= #Temp_Press_max,
	                                 PT:= T#30S,
	                                 Q=> #bar_max);
	  
	  
	END_REGION
	
END_FUNCTION_BLOCK

FUNCTION_BLOCK "Kontrola Hz w trybie awayjnym od barMax"
TITLE = Handing Oxygen Pressure Max
{ S7_Optimized_Access := 'TRUE' }
AUTHOR : rtecmer
VERSION : 0.1
//Sterowanie wydajnością invertera KDN w czasie wystąpienia alarmu od ciśnienia, przeciążenia
   VAR_INPUT 
      Value_Max : Bool;   // Znacznik Alarmowej wartości
      My_1Hz : Bool;
      Act_Hz : Real;   // Aktualne Hz przechwycone
      IsMotor2Set : Bool;   // Znacznik pierwszej pompy dodatkowej
      IsMotor3Set : Bool;   // Znacznik drugiej pompy dodatkowej
      IsMotor4Set : Bool;   // Znacznik drugiej pompy dodatkowej
      IsReadyinverter1 : Bool;   // Gotowość falownika 1
   END_VAR

   VAR_OUTPUT 
      Value_Manual_Hz : Real := 10.0;   // Wartość procentowa [%}  Hz zadawanych w trybie awaryjnym
      Rst_Motor2 : Bool;   // Znacznik wyłaczenia awayjnego dodatkowej pompy pierwszej
      Rst_Motor3 : Bool;   // Znacznik wyłaczenia awayjnego dodatkowej pompy drugiej
      Rst_Motor4 : Bool;   // Znacznik wyłaczenia awayjnego dodatkowej pompy drugiej
      Rst_Driver : Bool := false;   // Znacznik wyłaczenia awayjnego
   END_VAR

   VAR_TEMP 
      set_NewValue : Bool;
      index : Bool;
      CV : Int;
      load_cunt : Bool;
      tmp_Hz : Real;   // Wartość Hz zatrzaśnięta do obliczeń
      cnt_Hz : Real;   // Zmienna Hz do przeliczania w procesie sterowani podczas awarii
      mem_Triger_Alarm : Bool;   // Pamięć zbocza narastającego wytąpienia alarmu
   END_VAR

   VAR CONSTANT 
      PV : Int := 30;   // Wartość procentowa licznika ładowanego dla Generacji wartości [%] Hz
   END_VAR


BEGIN
	(*
	Kontrola wartości zadanej Hz w trybie pracy awaryjnej od max 
	ciśnienia  w przewodzie
	*)
	
	// Wyłączenie pompy pracującej w trybie sterowania awaryjnego bez falownika
	IF #IsReadyinverter1 = FALSE AND #Value_Max = TRUE THEN
	  // Ustaw znacznik wyłączenie awaryjnego
	  #Rst_Driver := TRUE;
	ELSE
	  #Rst_Driver := FALSE;
	END_IF;
	
	IF #IsReadyinverter1 THEN
	  // Blokowanie znacznika wyłączenia awaryjnego
	  #Rst_Driver := FALSE;
	END_IF;
	
	
	
	IF #Value_Max AND #IsMotor2Set AND #IsMotor3Set THEN
	  #Rst_Motor3 := TRUE;
	ELSE
	  #Rst_Motor3 := FALSE;
	END_IF;
	
	IF #Value_Max AND #IsMotor2Set AND (#IsMotor3Set = FALSE) THEN
	  #Rst_Motor2 := TRUE;
	ELSE
	  #Rst_Motor2 := FALSE;
	END_IF;
	
	IF #Value_Max AND #IsMotor4Set  THEN
	  #Rst_Motor4 := TRUE;
	ELSE
	  #Rst_Motor4 := FALSE;
	END_IF;
	
	
	IF "IEC_Counter_ControlAlarm_DB".CV > 55 THEN
	  // jeśli licznik doliczył do 55 to wyłaczenie zliczania
	  #load_cunt := FALSE;
	ELSE
	  #load_cunt := TRUE;
	  ;
	END_IF;
	
	
	REGION Licznik opóźnienie wstawienia nowej wartości Hz
	  
	  // Nalicznie nowej wartości Hz
	  IF #Value_Max THEN
	    #index := "My_1Hz";
	    "IEC_Counter_ControlAlarm_DB".CTD(CD:=#index,
	                                      LD:= #load_cunt,
	                                      PV:= #PV,
	                                      Q=> #set_NewValue,
	                                      CV=> #CV);
	
	    
	    
	    // Przekazanie nowej naliczonej wartości
	    IF #set_NewValue = FALSE AND #Value_Max AND  (#IsMotor2Set= FALSE) AND (#IsMotor3Set= FALSE)  THEN
	      // Przekazanie do bloku danych nowej wartości
	      
	        #Value_Manual_Hz := #CV;
	        "dbdane".tmp_Hz_ModeAlarm :=  #Value_Manual_Hz;
	        
	      ELSE
	        ;
	      END_IF;
	    END_IF;
	    
	  
	  IF #Value_Max = False THEN
	    #Value_Manual_Hz := 5.0;
	    
	  END_IF;
	    
	   
	  
	END_REGION
	
	
	
	
END_FUNCTION_BLOCK

FUNCTION "Błąd_Modbus_TCP" : Void
TITLE = Obsługa błedu komunikacji
{ S7_Optimized_Access := 'TRUE' }
AUTHOR : rtecmer
VERSION : 0.1
//Funkcja ubsługuje błędy komunikacji, czyści kody błędów po ponownym poprawnym nawiązaniu komunikacji modbus tcp 
   VAR_TEMP 
      reset : Bool;
      reset_1 : Bool;
   END_VAR


BEGIN
	(*
	//=============================================================================
	//(JZWiK S.A Radosław Tecmer)
	//(c)Copyright (2022) All Rights Reserved
	//-----------------------------------------------------------------------------
	//Testowane z:   (system docelowy z  FW 4.4)
	//Pakiet inżynierski:   TIA Portal (V16 Update 5)
	//Ograniczenia:  ( - )
	//Wymagania:  (minimalne S7-1200 CPU 1215C FW 4.2 .)
	//Funkcjonalnośc: (Funkcja ubsługuje błędy komunikacji, czyści kody błędów 
	                    po ponownym poprawnym nawiązaniu komunikacji modbus tcp )
	//-----------------------------------------------------------------------------
	//Zmainy wprowadzone:
	//Wersja  Data       Osoba wprowadzająca zmiany - ekspert
	//01.00.00 09.03.2022 (Tecmer Radosław - twórca) Pieresza wersja 01.00.00
	//=============================================================================
	*)
	
	(*
	REGION brak komunikacji z PLC - PLC 
	  // jeśli licznik kontroli komunikacji wskazuje brak komunikacji
	  IF "Dane_ComunicationControlHMI".tempCoordinationHMIRS5 > 23 OR  "db10organizacyjna".reset_modbus_TCP THEN
	    // restart modbus tcp
	    #reset := TRUE;
	    
	      "IEC_Timer_resetModbusTCP_DB".TP(IN:=#reset,
	                                       Q=> #reset_1,
	                                       PT:=T#2S);
	      IF #reset_1 THEN
	        // reset server modbus tcp 
	        "DISCONNECT_SERVER_1" := TRUE;
	        "DISCONNECT_SERVER_2" := TRUE;
	        "DISCONNECT_SERVER_3" := TRUE;
	        "DISCONNECT_SERVER_4" := TRUE;
	        "memRisingTriger_Data_1" := FALSE;
	        "memRisingTriger_Data_2" := FALSE;
	        "memRisingTriger_Data_3" := FALSE;
	        "memRisingTriger_Data_4" := FALSE;
	        "memRisingTriger_Data_5" := FALSE;
	        "memRisingTriger_Data_6" := FALSE;
	        "memRisingTriger_Data_7" := FALSE;
	        "memRisingTriger_Data_8" := FALSE;
	        "memRisingTriger_Data_9" := FALSE;
	        "memRisingTriger_Data_10" := FALSE;
	        "memRisingTriger_Data_11" := FALSE;
	        "memRisingTriger_Data_12" := FALSE;
	        "memRisingTriger_Data_13" := FALSE;
	        "memRisingTriger_Data_14" := FALSE;
	        "memRisingTriger_Data_15" := FALSE;
	        "memRisingTriger_Data_16" := FALSE;
	        "memTrig_Client_Receiving_1" := FALSE;
	        "memTrig_Client_Receiving_2" := FALSE;
	        "memTrig_Client_Receiving_3" := FALSE;
	        "memTrig_Client_Receiving_4" := FALSE;
	        "memTrig_Client_Receiving_5" := FALSE;
	        "memTrig_Client_Receiving_7" := FALSE;
	        "memTrig_Client_Receiving_8" := FALSE;
	        "memTrig_Client_Receiving_9" := FALSE;
	        "memTrig_Client_Receiving_10" := FALSE;
	        "memTrig_Client_Receiving_11" := FALSE;
	        "memTrig_Client_Receiving_12" := FALSE;
	        "memTrig_Client_Receiving_13" := FALSE;
	        "memTrig_Client_Receiving_14" := FALSE;
	        "memTrig_Client_Receiving_15" := FALSE;
	        "memTrig_Client_Receiving_16" := FALSE;
	        
	      ELSE
	        "DISCONNECT_SERVER_1" := FALSE;
	        "DISCONNECT_SERVER_2" := FALSE;
	        "DISCONNECT_SERVER_3" := FALSE;
	        "DISCONNECT_SERVER_4" := FALSE;
	        ;
	      END_IF;
	      
	    ELSE
	
	      
	    ;
	  END_IF;
	  
	  
	END_REGION
	
	*)
	
END_FUNCTION

FUNCTION_BLOCK "Inicjacja wartości startowych"
TITLE = Setup Write Parameters_KDN
{ S7_Optimized_Access := 'TRUE' }
AUTHOR : rtecmer
VERSION : 0.1
//Pobranie parametrów technologicznych i przekazanie ich do instancji "tags" w celu zachowania i wprowadzeni po resecie PLC
   VAR_TEMP 
      TimeHz_DInt : DInt;
   END_VAR


BEGIN
	(*
	//=============================================================================
	//(JZWiK S.A Radosław Tecmer)
	//(c)Copyright (2021) All Rights Reserved
	//-----------------------------------------------------------------------------
	//Testowane z:   (system docelowy z  FW 4.2)
	//Pakiet inżynierski:   TIA Portal (V14 Sp1 Update 9)
	//Ograniczenia:  ( - )
	//Wymagania:  (minimalne S7-1200 CPU 1214 FW 3.2 .)
	//Funkcjonalnośc: (Przekazanie warotości ostatnio wpisanych do instancji "tags 
	                   w celu przechowania danych. W czasie restartu CPU będą wczytywane
	                   do parametrów sterowania  )
	//-----------------------------------------------------------------------------
	//Zmainy wprowadzone:
	//Wersja  Data       Osoba wprowadzająca zmiany - ekspert
	//01.00.00 17.11.2021 (Tecmer Radosław - twórca) Pieresza wersja 01.00.00
	//=============================================================================
	*)
	
	
	REGION Sterowanie 
	  // przekazanie danych
	 
	  "dbtags_Sterowanie".SetupControlPompownia.Time_ONK1 := "db10organizacyjna".Time_ONK1;
	  "dbtags_Sterowanie".SetupControlPompownia.Time_ONK2 := "db10organizacyjna".Time_ONK2;
	  "dbtags_Sterowanie".SetupControlPompownia.Time_OFFK1:= "db10organizacyjna".Time_OFFK1;
	  "dbtags_Sterowanie".SetupControlPompownia.Time_OFFK2 := "db10organizacyjna".Time_OFFK2;
	  "dbtags_Sterowanie".SetupControlPompownia.TimeHz := "db10organizacyjna".TimeHz;
	  
	  //Czas oczekiwania na 50Hz 
	  "dbdane".TMR_Hz := DINT_TO_TIME(#TimeHz_DInt * "MS_TO_S");
	  
	  //Tryb pracy pompowni 
	  "dbtags_Sterowanie".SetupControlPompownia.Switch_Aut_Rem_Pompy := "dbzarządzanie".sterowanie_1.tryb_automat;
	  
	  //strategi pracy pompowni
	  "dbdane".Switch_model_control_P1P4 := "dbHoldRegSlave_to_MT101".instSygSter_1;
	  //strategia sterowaia zbiornikami
	  "dbdane".Switch_model_control_Tanks := "dbHoldRegSlave_to_MT101".instSygSter_2;
	  
	  //kasowanie alarmów napędów
	  "dbtags_Sterowanie"."Paramaetry _Zbiorniki".rez_alarm_napędów := "dbHoldRegSlave_to_MT101".instClearFault1;
	  
	  // zadane ciśnieniea
	  "dbtags_Sterowanie".SetupControlPompownia.set_barDN500_B5 := "dbHoldRegSlave_to_MT101".instSetbarDN500_B5;
	  "dbtags_Sterowanie".SetupControlPompownia.set_barDN225_B6 := "dbHoldRegSlave_to_MT101".instSetbarDN225_B6;
	  
	END_REGION
	
	REGION Z11 Z12 Status
	  // Przekazanie do instancji pamięci parametrów
	  IF %DB10.DBX118.7 = 1 THEN
	    // Gdy praca Auto ustaw
	    "dbtags_Sterowanie".SetupControlPompownia.Z11_Status := 33924;
	  ELSE
	    "dbtags_Sterowanie".SetupControlPompownia.Z11_Status := 0;
	  END_IF;
	  
	  IF %DB10.DBX120.7 = 1  THEN
	    // gdy praca Auto ustaw
	    "dbtags_Sterowanie".SetupControlPompownia.Z12_Status := 33924;
	  ELSE
	    "dbtags_Sterowanie".SetupControlPompownia.Z12_Status := 0;
	  END_IF;
	  
	 
	  
	  
	END_REGION
	
	REGION Parametry nastaw zbiorników 
	  // 
	  "dbtags_Sterowanie"."Paramaetry _Zbiorniki".set_poziom_napełniania:= "dbHold_RRG".set_poziom_napełniania ;
	  "dbtags_Sterowanie"."Paramaetry _Zbiorniki".set_poziom_opróżniania:= "dbHold_RRG".set_poziom_opróżniania ;
	  "dbtags_Sterowanie"."Paramaetry _Zbiorniki".set_strategia_sterowania := "dbHoldRegSlave_to_MT101".instSygSter_1;
	  "dbtags_Sterowanie"."Paramaetry _Zbiorniki".set_sterowanie_cyklem:= "dbHoldRegSlave_to_MT101".instSygSter_2 ;
	  "dbtags_Sterowanie"."Paramaetry _Zbiorniki".set_położenie_Z10:= "dbHold_RRG".set_położenie_Z10 ;
	  "dbtags_Sterowanie"."Paramaetry _Zbiorniki".set_bity_sterowania_napęami_1 := "dbHoldRegSlave_to_MT101".instControllDrivers_1;
	  "dbtags_Sterowanie"."Paramaetry _Zbiorniki".set_bity_sterowania_napęami_2 := "dbHoldRegSlave_to_MT101".instControllDrivers_2;
	  "dbtags_Sterowanie"."Paramaetry _Zbiorniki".set_bity_tryb_napędów_1 := "dbHoldRegSlave_to_MT101".instConrol_ManAut_1;
	  "dbtags_Sterowanie"."Paramaetry _Zbiorniki".set_bity_tryb_napędów_2 := "dbHoldRegSlave_to_MT101".instConrol_ManAut_2;
	  //Czasy
	  "dbtags_Sterowanie".Zbiorniki_Godziny.start_napełnianie.HOUR := "dbHoldRegSlave_to_MT101".instHourStart_Filling;
	  "dbtags_Sterowanie".Zbiorniki_Godziny.start_napełnianie.MINUTE := "dbHoldRegSlave_to_MT101".instMinutStart_Filling;
	  "dbtags_Sterowanie".Zbiorniki_Godziny.start_napełnianie.SECOND := 0;
	  
